(* IEC 61131-3 sources: fse/dataset/original (part 7) *)

(* ---- lb_claude_assisted_dd04b7ea0182_0007.st ---- *)
(*
This code implements a randomly grown symbolic expression:

((!(!(IN21 & (xor(xor(false, !(!((xor(xor(false, IN2), IN25)) | (!(IN9))))), ((IN33 & (xor(xor(IN17, IN40), IN11))) & (xor(xor(xor(xor(IN20, IN38), IN8), IN28 & IN33), IN19 & IN13))) & IN13))))) & IN25) & ((!((xor(xor(IN28, xor(xor((!(!(IN8 | IN21))) | ((!(IN47 | IN48)) | (!(IN15))), (!(IN9)) | ((xor(xor(IN49 & IN47, IN49 & IN24), IN46 | IN22)) | (!(IN28)))), !(((IN34 & IN44) & IN48) & IN26))), !(xor(xor(!((xor(xor(IN22, IN48), IN19)) | IN13), IN46), !((xor(xor(IN22, IN42), IN14)) | IN16))))) & ((((xor(xor((false | IN22) & (IN6 & IN36), (!(IN36)) & (IN1 & IN42)), IN21 & IN2)) | IN42) | IN48) | (!(IN36))))) & (IN15 | ((xor(xor(!(!(xor(xor((IN30 | IN11) | (IN43 & IN31), IN43 & (IN50 | IN12)), (IN13 & IN46) | (IN47 & IN18)))), ((IN47 | ((!(IN45)) & IN30)) & (xor(xor(xor(xor(IN6, IN1 & IN6), IN47), xor(xor(IN1 | IN29, IN33), false)), IN35))) | (xor(xor(((!(IN21)) | (!(IN25))) & (IN46 & (IN9 | IN19)), xor(xor(!(IN12 | IN11), xor(xor(IN8 & IN17, IN35 & IN20), xor(xor(IN38, IN14), IN18))), IN36 | (IN49 | IN43))), xor(xor((IN5 & IN20) & (xor(xor(IN20, IN17), IN15)), (xor(xor(IN2, IN24), IN37)) & IN6), IN18 & (IN41 | IN4))))), !(xor(xor(IN3, IN35), (xor(xor(IN29 & IN48, xor(xor(IN41, IN30), IN24)), IN15 | IN43)) | ((!(IN29)) | (false | IN42)))))) & (!(!(IN21 | (((!(IN38)) | (IN48 | IN49)) | IN16)))))))

*)

FUNCTION_BLOCK F_CollectInput
  VAR_IN_OUT
      Data : ARRAY[1..50] OF BOOL;
  END_VAR
  VAR_INPUT
      TICK  : BOOL := 0;
      IN1   : BOOL := 0;
      IN2   : BOOL := 0;
      IN3   : BOOL := 0;
      IN4   : BOOL := 0;
      IN5   : BOOL := 0;
      RESET : BOOL := FALSE;
  END_VAR
  VAR_OUTPUT
      Finished : BOOL;
  END_VAR
  VAR
      j    : USINT := 1;
      tock : BOOL  := 0;
  END_VAR
  IF NOT RESET AND tock = NOT TICK THEN
      Data[j]   := IN1;
      Data[j+1] := IN2;
      Data[j+2] := IN3;
      Data[j+3] := IN4;
      Data[j+4] := IN5;
      j := j + 5;
      tock := TICK;
  ELSE
      j := 1;
      tock := 0;
  END_IF;
  Finished := (j > 50);
END_FUNCTION_BLOCK

PROGRAM Boiler
  VAR
    Data  : ARRAY[1..50] OF BOOL;
    Ready : BOOL;
    CollectInput : F_CollectInput;
  END_VAR
  VAR
    TICK     AT %IX1.0 : BOOL;
    IN1      AT %IX0.3 : BOOL;
    IN2      AT %IX0.4 : BOOL;
    IN3      AT %IX0.5 : BOOL;
    IN4      AT %IX0.6 : BOOL;
    IN5      AT %IX0.7 : BOOL;
    OutReady AT %QX0.0 : BOOL := FALSE;
    FeedNext AT %QX0.1 : BOOL := FALSE;
    Out      AT %QX0.2 : BOOL;
  END_VAR
  CollectInput(TICK:=TICK, IN1:=IN1, IN2:=IN2, IN3:=IN3, IN4:=IN4, IN5:=IN5);
  Ready := CollectInput.Finished;
  FeedNext := 1;
  IF Ready THEN
    Out := (((NOT (NOT (Data[21] AND ((FALSE XOR (NOT (NOT (((FALSE XOR Data[2]) XOR Data[25]) OR (NOT Data[9]))))) XOR (((Data[33] AND ((Data[17] XOR Data[40]) XOR Data[11])) AND ((((Data[20] XOR Data[38]) XOR Data[8]) XOR (Data[28] AND Data[33])) XOR (Data[19] AND Data[13]))) AND Data[13]))))) AND Data[25]) AND ((NOT (((Data[28] XOR ((((NOT (NOT (Data[8] OR Data[21]))) OR ((NOT (Data[47] OR Data[48])) OR (NOT Data[15]))) XOR ((NOT Data[9]) OR ((((Data[49] AND Data[47]) XOR (Data[49] AND Data[24])) XOR (Data[46] OR Data[22])) OR (NOT Data[28])))) XOR (NOT (((Data[34] AND Data[44]) AND Data[48]) AND Data[26])))) XOR (NOT (((NOT (((Data[22] XOR Data[48]) XOR Data[19]) OR Data[13])) XOR Data[46]) XOR (NOT (((Data[22] XOR Data[42]) XOR Data[14]) OR Data[16]))))) AND (((((((FALSE OR Data[22]) AND (Data[6] AND Data[36])) XOR ((NOT Data[36]) AND (Data[1] AND Data[42]))) XOR (Data[21] AND Data[2])) OR Data[42]) OR Data[48]) OR (NOT Data[36])))) AND (Data[15] OR ((((NOT (NOT ((((Data[30] OR Data[11]) OR (Data[43] AND Data[31])) XOR (Data[43] AND (Data[50] OR Data[12]))) XOR ((Data[13] AND Data[46]) OR (Data[47] AND Data[18]))))) XOR (((Data[47] OR ((NOT Data[45]) AND Data[30])) AND ((((Data[6] XOR (Data[1] AND Data[6])) XOR Data[47]) XOR (((Data[1] OR Data[29]) XOR Data[33]) XOR FALSE)) XOR Data[35])) OR (((((NOT Data[21]) OR (NOT Data[25])) AND (Data[46] AND (Data[9] OR Data[19]))) XOR (((NOT (Data[12] OR Data[11])) XOR (((Data[8] AND Data[17]) XOR (Data[35] AND Data[20])) XOR ((Data[38] XOR Data[14]) XOR Data[18]))) XOR (Data[36] OR (Data[49] OR Data[43])))) XOR ((((Data[5] AND Data[20]) AND ((Data[20] XOR Data[17]) XOR Data[15])) XOR (((Data[2] XOR Data[24]) XOR Data[37]) AND Data[6])) XOR (Data[18] AND (Data[41] OR Data[4])))))) XOR (NOT ((Data[3] XOR Data[35]) XOR ((((Data[29] AND Data[48]) XOR ((Data[41] XOR Data[30]) XOR Data[24])) XOR (Data[15] OR Data[43])) OR ((NOT Data[29]) OR (FALSE OR Data[42])))))) AND (NOT (NOT (Data[21] OR (((NOT Data[38]) OR (Data[48] OR Data[49])) OR Data[16]))))))));
    OutReady := 1;
    CollectInput(RESET:=TRUE);
  END_IF;
END_PROGRAM

CONFIGURATION Config0
  RESOURCE Res0 ON PLC
    TASK task0(INTERVAL := T#20ms,PRIORITY := 0);
    PROGRAM instance0 WITH task0 : Boiler;
  END_RESOURCE
END_CONFIGURATION

(* ---- lb_claude_assisted_ddda264e743a_0020.st ---- *)
FUNCTION_BLOCK T_PLC_MS_block
	VAR_OUTPUT
		T_PLC_MS :	UDINT;
	END_VAR

	VAR_EXTERNAL
		PLC_TICKS_PER_SEC :	INT;
		PLC_SYS_TICK_CNT :	DINT;
	END_VAR

	VAR
		debug :	BOOL;(*Debug-Mode ON / OFF*)
		N :	INT;(*Debug-Faktor*)
		Offset :	UDINT;(*Debug-Offset*)
		temp :	DWORD := DWORD#1;(*Debug-Offset*)
		mode :	BOOL;(*modus*)
		faktor :	UDINT;(*Systemtakt-Faktor*)
		init :	BOOL;
		v_plc_ticks_per_sec :	UDINT;
		base :	UDINT := UDINT#1000;
	END_VAR

	IF init = FALSE THEN
		v_plc_ticks_per_sec := INT_TO_UDINT(PLC_TICKS_PER_SEC);
		IF v_plc_ticks_per_sec = UDINT#1024 THEN
			faktor := UDINT#1;
			mode := FALSE;
		ELSIF v_plc_ticks_per_sec > UDINT#0 THEN
			IF v_plc_ticks_per_sec <= base THEN
				faktor := base / v_plc_ticks_per_sec;
				mode := FALSE;
			ELSE
				faktor := v_plc_ticks_per_sec / base;
				mode := TRUE;
			END_IF;
		ELSE
			faktor := UDINT#1;
		END_IF;
		init := TRUE;
	END_IF;

	IF mode THEN
		T_PLC_MS := DINT_TO_UDINT(PLC_SYS_TICK_CNT) / faktor;
	ELSE
		T_PLC_MS := DINT_TO_UDINT(PLC_SYS_TICK_CNT) * faktor;
	END_IF;

	IF debug THEN
		T_PLC_MS := (DWORD_TO_UDINT(SHL(UDINT_TO_DWORD(T_PLC_MS),N) OR SHL(temp,N)) - UDINT#1) + Offset;
	END_IF;
END_FUNCTION_BLOCK

FUNCTION TIME_TO_UDINT2:UDINT
	VAR_INPUT
		X :	TIME;
	END_VAR

	TIME_TO_UDINT2 := DINT_TO_UDINT(TIME_TO_DINT(X));
END_FUNCTION

FUNCTION_BLOCK TUNE2_Block

	VAR_INPUT
		SET :	BOOL;
		SU :	BOOL;
		SD :	BOOL;
		FU :	BOOL;
		FD :	BOOL;
		RST :	BOOL;
		SS :	REAL := 0.1;
		FS :	REAL := 5.0;
		LIMIT_L :	REAL;
		LIMIT_H :	REAL := 100.0;
		RST_VAL :	REAL;
		SET_VAL :	REAL := 100.0;
		TR :	TIME := T#500ms;
		S1 :	REAL := 2.0;
		S2 :	REAL := 10.0;
	END_VAR

	VAR_OUTPUT
		Y :	REAL;
	END_VAR

	VAR
		tx :	UDINT;
		start :	UDINT;
		state :	INT;
		in :	BOOL;
		step2 :	REAL;
		speed :	REAL;
		Y_start :	REAL;
		T_PLC_MS :	T_PLC_MS_block;
	END_VAR

	T_PLC_MS();
	tx:= T_PLC_MS.T_PLC_MS;

	IF rst THEN
		Y := RST_val;
		state := 0;
	ELSIF set THEN
		Y := SET_val;
		state := 0;
	ELSIF state > 0 THEN
		CASE state OF
			1 :
				in := su;
			2 :
				in := sd;
			3 :
				in := fu;
			4 :
				in := fd;
		END_CASE;
		IF NOT in AND tx - start <= TIME_TO_UDINT2(TR) THEN
			Y := Y_start + step2;
			state := 0;
		ELSIF in AND tx - start >= TIME_TO_UDINT2(TR) THEN
			Y := Y_start + UDINT_TO_REAL(tx - start - TIME_TO_UDINT2(TR)) * speed;
		ELSIF NOT in THEN
			state := 0;
		END_IF;
	ELSIF su THEN
		state := 1;
		start := tx;
		step2 := ss;
		speed := s1 * 1.0E-3;
		Y_start := Y;
	ELSIF sd THEN
		state := 2;
		start := tx;
		step2 := -ss;
		speed := -s1 * 1.0E-3;
		Y_start := Y;
	ELSIF fu THEN
		state := 3;
		start := tx;
		step2 := fs;
		speed := s2 * 1.0E-3;
		y_start := Y;
	ELSIF fd THEN
		state := 4;
		start := tx;
		step2 := -fs;
		speed := -s2 * 1.0E-3;
		y_start := Y;
	END_IF;
END_FUNCTION_BLOCK

PROGRAM program0
  	VAR
		SET :	BOOL;
		SU :	BOOL;
		SD :	BOOL;
		FU :	BOOL;
		FD :	BOOL;
		RST :	BOOL;
		SS :	REAL;
		FS :	REAL;
		LIMIT_L :	REAL;
		LIMIT_H :	REAL;
		RST_VAL :	REAL;
		SET_VAL :	REAL;
		TR :	TIME ;
		S1 :	REAL;
		S2 :	REAL;
		Y :	REAL;
		func_block : TUNE2_Block;
  	END_VAR
	func_block.SET := SET;
	func_block.SU := SU;
	func_block.SD := SD;
	func_block.FU := FU;
	func_block.FD := FD;
	func_block.RST := RST;
	func_block.SS:= SS;
	func_block.FS := FS;
	func_block.LIMIT_L := LIMIT_L;
	func_block.LIMIT_H := LIMIT_H;
	func_block.RST_VAL := RST_VAL;
	func_block.SET_VAL := SET_VAL;
	func_block.TR := TR;
	func_block.S1 := S1;
	func_block.S2 := S2;
	func_block();
	Y := func_block.Y;
END_PROGRAM

CONFIGURATION Config0
	VAR_GLOBAL
		PLC_TICKS_PER_SEC :	INT;
		PLC_SYS_TICK_CNT :	DINT;
	END_VAR

	RESOURCE Res0 ON PLC
		TASK task0(INTERVAL := T#20ms,PRIORITY := 0);
		PROGRAM instance0 WITH task0 : program0;
	END_RESOURCE
END_CONFIGURATION

(* ---- lb_claude_assisted_def584e78dd9_0028.st ---- *)
(*
This code implements a randomly grown symbolic expression:

((xor(xor(!(IN17), IN3), IN42 & (!(!((!(xor(xor(IN42 & IN8, IN18), IN49))) | (!(IN32))))))) & ((!(!((IN47 | (IN12 & (xor(xor(!(IN9), IN41 & IN17), IN45)))) & (xor(xor(IN6 & (IN23 | (IN31 | IN44)), xor(xor((!(IN32)) & (!(IN23)), IN42 & (IN50 | IN34)), xor(xor(!(IN34), !(IN32)), IN15))), xor(xor(IN33, xor(xor(IN45 & IN5, IN11 & IN16), IN3 | IN4)), !(!(IN15)))))))) & (((xor(xor(((xor(xor(IN50 | IN14, IN46 & IN40), xor(xor(IN3, IN41), IN9))) & (IN22 & IN28)) | (xor(xor(IN41 | (IN26 & IN10), xor(xor(IN42 & IN12, xor(xor(IN32, IN46), IN35)), IN1 & IN11)), xor(xor(xor(xor(IN43, IN19), IN38), IN27 | IN21), !(IN10)))), !(xor(xor((xor(xor(IN7, IN50), IN1)) | IN6, (IN35 & IN3) | (!(IN28))), xor(xor(IN7 & IN16, IN37 | IN33), IN11)))), (!((!(IN25)) | (!(IN41)))) & ((!(IN33 & true)) & (!(!(IN5)))))) & (xor(xor(IN12, !(IN17)), (((!(IN28)) & (xor(xor(IN4, IN22), IN12))) | ((IN4 & IN38) & IN37)) | true))) | IN6))) & (xor(xor(!(IN24), xor(xor(!((xor(xor(IN48 | (!((IN17 & IN14) | IN31)), (xor(xor(true, xor(xor(xor(xor(IN16, IN16), IN17), !(IN23)), IN2)), (!(IN45)) | (xor(xor(IN31, IN48), IN25)))) & (!(xor(xor(IN6, IN41 & IN37), IN38)))), (IN26 | ((IN7 & IN2) | (IN17 | false))) & (xor(xor(IN42 & (IN28 | IN44), (IN16 & IN26) | (IN21 | IN13)), (IN11 & IN4) | (IN48 | IN47))))) & ((!(false & ((xor(xor(IN20, IN8), IN2)) | (IN36 & IN18)))) & IN47)), xor(xor(((false & (xor(xor(xor(xor(IN27 | IN30, xor(xor(IN23, IN27), IN7)), IN21), !(IN50)), (!(IN35)) & (xor(xor(IN21, IN7), IN17))))) | ((((IN9 | IN5) | (xor(xor(IN46, IN31), IN33))) | IN14) | IN32)) | (((!(IN19)) & IN21) & (!((!(IN44 & IN26)) | IN42))), xor(xor(!(IN34), (IN31 | (xor(xor(IN20, IN9), IN30))) | (xor(xor(IN21, xor(xor((IN29 | IN5) | (IN10 & IN14), xor(xor(IN41 & IN34, xor(xor(IN20, IN4), IN29)), IN29 & IN17)), IN39 | (IN7 & IN43))), ((!(IN40)) | IN50) | (!(IN17))))), xor(xor(xor(xor(IN31, IN24), ((IN30 | IN5) & (!(IN48))) | ((xor(xor(IN16, IN13), IN34)) & (!(IN16)))), (xor(xor(IN29 | IN25, xor(xor(xor(xor(IN20, IN40), IN9), IN26 | IN20), IN43 | IN32)), (xor(xor(IN35, IN6), IN33)) | (IN30 | IN7))) & (((true | IN15) | (IN46 | IN5)) | ((xor(xor(IN20, IN39), IN5)) | (IN48 | IN20)))), ((!(IN11 & IN1)) | ((xor(xor(IN5, IN25), IN49)) | (IN3 & IN43))) | (!(xor(xor(IN22, xor(xor(IN40, IN26), IN7)), xor(xor(IN10, IN10), IN44))))))), !(xor(xor(!(xor(xor((!(IN32)) | (xor(xor(IN28, IN4), IN11)), (IN7 | IN49) & (IN19 | IN17)), xor(xor(xor(xor(IN50, IN4), IN7), !(IN25)), !(IN10)))), (xor(xor(IN18 & (IN23 | IN36), xor(xor(IN36 | false, IN31 | IN19), IN15 & IN5)), !(IN41))) | (!(!(xor(xor(IN34, IN8), true))))), IN10 & (((IN39 & IN8) | (xor(xor(IN37, IN1), IN46))) | ((xor(xor(IN21, IN1), IN16)) | (false | IN1))))))), IN25 & (IN31 & (IN20 & IN46)))), IN38 | (!(IN32))))

*)

FUNCTION_BLOCK F_CollectInput
  VAR_IN_OUT
      Data : ARRAY[1..50] OF BOOL;
  END_VAR
  VAR_INPUT
      TICK  : BOOL := 0;
      IN1   : BOOL := 0;
      IN2   : BOOL := 0;
      IN3   : BOOL := 0;
      IN4   : BOOL := 0;
      IN5   : BOOL := 0;
      RESET : BOOL := FALSE;
  END_VAR
  VAR_OUTPUT
      Finished : BOOL;
  END_VAR
  VAR
      j    : USINT := 1;
      tock : BOOL  := 0;
  END_VAR
  IF NOT RESET AND tock = NOT TICK THEN
      Data[j]   := IN1;
      Data[j+1] := IN2;
      Data[j+2] := IN3;
      Data[j+3] := IN4;
      Data[j+4] := IN5;
      j := j + 5;
      tock := TICK;
  ELSE
      j := 1;
      tock := 0;
  END_IF;
  Finished := (j > 50);
END_FUNCTION_BLOCK

PROGRAM Boiler
  VAR
    Data  : ARRAY[1..50] OF BOOL;
    Ready : BOOL;
    CollectInput : F_CollectInput;
  END_VAR
  VAR
    TICK     AT %IX1.0 : BOOL;
    IN1      AT %IX0.3 : BOOL;
    IN2      AT %IX0.4 : BOOL;
    IN3      AT %IX0.5 : BOOL;
    IN4      AT %IX0.6 : BOOL;
    IN5      AT %IX0.7 : BOOL;
    OutReady AT %QX0.0 : BOOL := FALSE;
    FeedNext AT %QX0.1 : BOOL := FALSE;
    Out      AT %QX0.2 : BOOL;
  END_VAR
  CollectInput(TICK:=TICK, IN1:=IN1, IN2:=IN2, IN3:=IN3, IN4:=IN4, IN5:=IN5);
  Ready := CollectInput.Finished;
  FeedNext := 1;
  IF Ready THEN
    Out := (((((NOT Data[17]) XOR Data[3]) XOR (Data[42] AND (NOT (NOT ((NOT (((Data[42] AND Data[8]) XOR Data[18]) XOR Data[49])) OR (NOT Data[32])))))) AND ((NOT (NOT ((Data[47] OR (Data[12] AND (((NOT Data[9]) XOR (Data[41] AND Data[17])) XOR Data[45]))) AND (((Data[6] AND (Data[23] OR (Data[31] OR Data[44]))) XOR ((((NOT Data[32]) AND (NOT Data[23])) XOR (Data[42] AND (Data[50] OR Data[34]))) XOR (((NOT Data[34]) XOR (NOT Data[32])) XOR Data[15]))) XOR ((Data[33] XOR (((Data[45] AND Data[5]) XOR (Data[11] AND Data[16])) XOR (Data[3] OR Data[4]))) XOR (NOT (NOT Data[15]))))))) AND (((((((((Data[50] OR Data[14]) XOR (Data[46] AND Data[40])) XOR ((Data[3] XOR Data[41]) XOR Data[9])) AND (Data[22] AND Data[28])) OR (((Data[41] OR (Data[26] AND Data[10])) XOR (((Data[42] AND Data[12]) XOR ((Data[32] XOR Data[46]) XOR Data[35])) XOR (Data[1] AND Data[11]))) XOR ((((Data[43] XOR Data[19]) XOR Data[38]) XOR (Data[27] OR Data[21])) XOR (NOT Data[10])))) XOR (NOT (((((Data[7] XOR Data[50]) XOR Data[1]) OR Data[6]) XOR ((Data[35] AND Data[3]) OR (NOT Data[28]))) XOR (((Data[7] AND Data[16]) XOR (Data[37] OR Data[33])) XOR Data[11])))) XOR ((NOT ((NOT Data[25]) OR (NOT Data[41]))) AND ((NOT (Data[33] AND TRUE)) AND (NOT (NOT Data[5]))))) AND ((Data[12] XOR (NOT Data[17])) XOR ((((NOT Data[28]) AND ((Data[4] XOR Data[22]) XOR Data[12])) OR ((Data[4] AND Data[38]) AND Data[37])) OR TRUE))) OR Data[6]))) AND (((NOT Data[24]) XOR (((NOT ((((Data[48] OR (NOT ((Data[17] AND Data[14]) OR Data[31]))) XOR (((TRUE XOR ((((Data[16] XOR Data[16]) XOR Data[17]) XOR (NOT Data[23])) XOR Data[2])) XOR ((NOT Data[45]) OR ((Data[31] XOR Data[48]) XOR Data[25]))) AND (NOT ((Data[6] XOR (Data[41] AND Data[37])) XOR Data[38])))) XOR ((Data[26] OR ((Data[7] AND Data[2]) OR (Data[17] OR FALSE))) AND (((Data[42] AND (Data[28] OR Data[44])) XOR ((Data[16] AND Data[26]) OR (Data[21] OR Data[13]))) XOR ((Data[11] AND Data[4]) OR (Data[48] OR Data[47]))))) AND ((NOT (FALSE AND (((Data[20] XOR Data[8]) XOR Data[2]) OR (Data[36] AND Data[18])))) AND Data[47]))) XOR (((((FALSE AND (((((Data[27] OR Data[30]) XOR ((Data[23] XOR Data[27]) XOR Data[7])) XOR Data[21]) XOR (NOT Data[50])) XOR ((NOT Data[35]) AND ((Data[21] XOR Data[7]) XOR Data[17])))) OR ((((Data[9] OR Data[5]) OR ((Data[46] XOR Data[31]) XOR Data[33])) OR Data[14]) OR Data[32])) OR (((NOT Data[19]) AND Data[21]) AND (NOT ((NOT (Data[44] AND Data[26])) OR Data[42])))) XOR (((NOT Data[34]) XOR ((Data[31] OR ((Data[20] XOR Data[9]) XOR Data[30])) OR ((Data[21] XOR ((((Data[29] OR Data[5]) OR (Data[10] AND Data[14])) XOR (((Data[41] AND Data[34]) XOR ((Data[20] XOR Data[4]) XOR Data[29])) XOR (Data[29] AND Data[17]))) XOR (Data[39] OR (Data[7] AND Data[43])))) XOR (((NOT Data[40]) OR Data[50]) OR (NOT Data[17]))))) XOR ((((Data[31] XOR Data[24]) XOR (((Data[30] OR Data[5]) AND (NOT Data[48])) OR (((Data[16] XOR Data[13]) XOR Data[34]) AND (NOT Data[16])))) XOR ((((Data[29] OR Data[25]) XOR ((((Data[20] XOR Data[40]) XOR Data[9]) XOR (Data[26] OR Data[20])) XOR (Data[43] OR Data[32]))) XOR (((Data[35] XOR Data[6]) XOR Data[33]) OR (Data[30] OR Data[7]))) AND (((TRUE OR Data[15]) OR (Data[46] OR Data[5])) OR (((Data[20] XOR Data[39]) XOR Data[5]) OR (Data[48] OR Data[20]))))) XOR (((NOT (Data[11] AND Data[1])) OR (((Data[5] XOR Data[25]) XOR Data[49]) OR (Data[3] AND Data[43]))) OR (NOT ((Data[22] XOR ((Data[40] XOR Data[26]) XOR Data[7])) XOR ((Data[10] XOR Data[10]) XOR Data[44]))))))) XOR (NOT (((NOT ((((NOT Data[32]) OR ((Data[28] XOR Data[4]) XOR Data[11])) XOR ((Data[7] OR Data[49]) AND (Data[19] OR Data[17]))) XOR ((((Data[50] XOR Data[4]) XOR Data[7]) XOR (NOT Data[25])) XOR (NOT Data[10])))) XOR ((((Data[18] AND (Data[23] OR Data[36])) XOR (((Data[36] OR FALSE) XOR (Data[31] OR Data[19])) XOR (Data[15] AND Data[5]))) XOR (NOT Data[41])) OR (NOT (NOT ((Data[34] XOR Data[8]) XOR TRUE))))) XOR (Data[10] AND (((Data[39] AND Data[8]) OR ((Data[37] XOR Data[1]) XOR Data[46])) OR (((Data[21] XOR Data[1]) XOR Data[16]) OR (FALSE OR Data[1])))))))) XOR (Data[25] AND (Data[31] AND (Data[20] AND Data[46]))))) XOR (Data[38] OR (NOT Data[32]))));
    OutReady := 1;
    CollectInput(RESET:=TRUE);
  END_IF;
END_PROGRAM

CONFIGURATION Config0
  RESOURCE Res0 ON PLC
    TASK task0(INTERVAL := T#20ms,PRIORITY := 0);
    PROGRAM instance0 WITH task0 : Boiler;
  END_RESOURCE
END_CONFIGURATION

(* ---- lb_claude_assisted_df27abd0aee2_0074.st ---- *)
FUNCTION_BLOCK EQ_0
  VAR_INPUT
    IN1 : DINT;
    IN2 : DINT;
  END_VAR
  VAR_OUTPUT
    OUT : BOOL;
  END_VAR
  VAR
    i : INT;
    mytimer : TON;
  END_VAR

  OUT:=FALSE;
  IF IN1=IN2 then
    OUT:=TRUE;
  END_IF;

  mytimer(IN := TRUE, PT := t#8000ms);
  i:=0;
  IF mytimer.Q = TRUE then
     WHILE i<4 do
      OUT:=TRUE;
    End_WHILE;
  End_IF;

END_FUNCTION_BLOCK

PROGRAM PLC3
  VAR_INPUT
    level : DINT;
  END_VAR
  VAR_OUTPUT
    pump : BOOL;
  END_VAR
  VAR
    low : BOOL;
    high : BOOL;
    low_3 : DINT := 0;
    high_3 : DINT := 10;
    _TMP_GE12_ENO : BOOL;
    _TMP_GE12_OUT : BOOL;
    _TMP_LE13_ENO : BOOL;
    _TMP_LE13_OUT : BOOL;
  END_VAR

  _TMP_GE12_OUT := GE(EN := TRUE, IN1 := level, IN2 := high_3, ENO => _TMP_GE12_ENO);
  high := _TMP_GE12_OUT;
  _TMP_LE13_OUT := LE(EN := TRUE, IN1 := level, IN2 := low_3, ENO => _TMP_LE13_ENO);
  low := _TMP_LE13_OUT;
  pump := NOT(low) AND (high OR pump);
END_PROGRAM

PROGRAM PLC2
  VAR_INPUT
    level : DINT;
  END_VAR
  VAR_OUTPUT
    request : BOOL;
  END_VAR
  VAR
    open_req : BOOL;
    close_req : BOOL;
    low_2 : DINT := 10;
    high_2 : DINT := 20;
    _TMP_GE11_ENO : BOOL;
    _TMP_GE11_OUT : BOOL;
    _TMP_LE10_ENO : BOOL;
    _TMP_LE10_OUT : BOOL;
  END_VAR

  _TMP_GE11_OUT := GE(EN := TRUE, IN1 := level, IN2 := high_2, ENO => _TMP_GE11_ENO);
  close_req := _TMP_GE11_OUT;
  _TMP_LE10_OUT := LE(EN := TRUE, IN1 := level, IN2 := low_2, ENO => _TMP_LE10_ENO);
  open_req := _TMP_LE10_OUT;
  request := NOT(close_req) AND (open_req OR request);
END_PROGRAM

PROGRAM PLC1
  VAR_INPUT
    level : DINT;
    request : DINT;
  END_VAR
  VAR_OUTPUT
    pumps : BOOL;
    valve : BOOL;
  END_VAR
  VAR
    low : BOOL;
    high : BOOL;
    open_req : BOOL;
    close_req : BOOL;
    low_1 : DINT := 40;
    high_1 : DINT := 80;
    EQ_00 : EQ_0;
    _TMP_EQ24_ENO : BOOL;
    _TMP_EQ24_OUT : BOOL;
    _TMP_LE3_ENO : BOOL;
    _TMP_LE3_OUT : BOOL;
    _TMP_GE7_ENO : BOOL;
    _TMP_GE7_OUT : BOOL;
  END_VAR

  EQ_00(EN := TRUE, IN1 := request, IN2 := 1);
  open_req := EQ_00.OUT;
  _TMP_EQ24_OUT := EQ(EN := TRUE, IN1 := request, IN2 := 0, ENO => _TMP_EQ24_ENO);
  close_req := _TMP_EQ24_OUT;
  pumps := NOT(high) AND (low OR pumps);
  valve := NOT(close_req) AND (valve OR open_req AND NOT(low));
  _TMP_LE3_OUT := LE(EN := TRUE, IN1 := level, IN2 := low_1, ENO => _TMP_LE3_ENO);
  low := _TMP_LE3_OUT;
  _TMP_GE7_OUT := GE(EN := TRUE, IN1 := level, IN2 := high_1, ENO => _TMP_GE7_ENO);
  high := _TMP_GE7_OUT;
END_PROGRAM

CONFIGURATION Config0

  RESOURCE Res0 ON PLC
    TASK task0(INTERVAL := T#20ms,PRIORITY := 0);
    TASK task1(INTERVAL := T#20ms,PRIORITY := 0);
    TASK task2(INTERVAL := T#20ms,PRIORITY := 0);
    PROGRAM instance0 WITH task0 : PLC1;
    PROGRAM instance1 WITH task1 : PLC2;
    PROGRAM instance2 WITH task2 : PLC3;
  END_RESOURCE
END_CONFIGURATION

(* ---- lb_claude_assisted_e1afd5a5507c_0051.st ---- *)
(*
This code implements a randomly grown symbolic expression:

(IN29 | (((!(IN27)) | (xor(xor(!(xor(xor(!((!(IN8)) & IN9), xor(xor(xor(xor(xor(xor(IN14, IN9), IN41), xor(xor(IN8, IN28), false)), xor(xor(IN9, IN9), IN2)), !(xor(xor(IN2, IN5), IN41))), (!(IN28)) & (xor(xor(IN12, IN39), IN7)))), IN36)), xor(xor(true, !(((IN30 | IN20) | IN9) & IN3)), xor(xor(false, (!(IN31)) | (xor(xor(IN41 | IN5, IN49 & IN1), !(IN13)))), xor(xor((IN28 | IN50) | (!(IN16)), (xor(xor(IN42, IN4), IN6)) | (xor(xor(IN38, IN42), IN36))), (xor(xor(IN46, IN18), IN35)) & (IN39 & IN11))))), IN39))) & (!(xor(xor(IN22 | ((!(xor(xor(IN21, IN5), IN41 & IN1))) | (xor(xor(xor(xor(IN15 | IN13, IN38 | IN6), !(IN1)), IN29), IN48))), IN18), IN3))))) | (!(!((((IN22 | (xor(xor(!(xor(xor(IN30, false), IN5)), !(IN14 | IN3)), !(IN48)))) | ((((!(IN28)) & (xor(xor(IN29, IN6), IN15))) & ((IN8 & IN49) | IN23)) & (((IN12 & IN1) | (xor(xor(IN43, IN5), IN47))) & ((!(IN33)) | (true | IN20))))) & ((!(IN50 | (!(IN5 | IN30)))) & IN40)) & (xor(xor((xor(xor((xor(xor(xor(xor(IN22, IN30), IN10), IN50), IN23 | IN47)) | (IN1 & (xor(xor(IN46, IN29), IN24))), IN24), ((IN2 & IN18) | (IN26 | IN47)) | ((!(IN19)) & IN35))) | ((IN33 & (!(IN25 | IN20))) | (xor(xor((xor(xor(IN40, IN13), IN19)) & (xor(xor(IN2, IN37), IN10)), (IN49 | IN40) & IN19), (xor(xor(IN25, IN24), IN14)) & (IN22 & IN32)))), (!(!((xor(xor(IN42, IN8), IN1)) & (!(IN42))))) & ((!(IN23 & IN19)) | ((!(IN29 & IN50)) & (!(IN8 & IN35))))), !(xor(xor(xor(xor((IN29 & IN22) & (!(IN14)), (IN32 & IN20) & (xor(xor(IN7, IN24), IN7))), (true & IN45) | (IN31 | IN44)), (xor(xor(!(IN45), IN35 | IN9), IN40 | IN3)) | ((xor(xor(IN5, IN37), IN27)) | (xor(xor(IN25, IN45), IN32)))), (false & (IN9 | IN18)) | (xor(xor(IN8, xor(xor(IN10, IN26), IN25)), !(IN39))))))))))

*)

FUNCTION_BLOCK F_CollectInput
  VAR_IN_OUT
      Data : ARRAY[1..50] OF BOOL;
  END_VAR
  VAR_INPUT
      TICK  : BOOL := 0;
      IN1   : BOOL := 0;
      IN2   : BOOL := 0;
      IN3   : BOOL := 0;
      IN4   : BOOL := 0;
      IN5   : BOOL := 0;
      RESET : BOOL := FALSE;
  END_VAR
  VAR_OUTPUT
      Finished : BOOL;
  END_VAR
  VAR
      j    : USINT := 1;
      tock : BOOL  := 0;
  END_VAR
  IF NOT RESET AND tock = NOT TICK THEN
      Data[j]   := IN1;
      Data[j+1] := IN2;
      Data[j+2] := IN3;
      Data[j+3] := IN4;
      Data[j+4] := IN5;
      j := j + 5;
      tock := TICK;
  ELSE
      j := 1;
      tock := 0;
  END_IF;
  Finished := (j > 50);
END_FUNCTION_BLOCK

PROGRAM Boiler
  VAR
    Data  : ARRAY[1..50] OF BOOL;
    Ready : BOOL;
    CollectInput : F_CollectInput;
  END_VAR
  VAR
    TICK     AT %IX1.0 : BOOL;
    IN1      AT %IX0.3 : BOOL;
    IN2      AT %IX0.4 : BOOL;
    IN3      AT %IX0.5 : BOOL;
    IN4      AT %IX0.6 : BOOL;
    IN5      AT %IX0.7 : BOOL;
    OutReady AT %QX0.0 : BOOL := FALSE;
    FeedNext AT %QX0.1 : BOOL := FALSE;
    Out      AT %QX0.2 : BOOL;
  END_VAR
  CollectInput(TICK:=TICK, IN1:=IN1, IN2:=IN2, IN3:=IN3, IN4:=IN4, IN5:=IN5);
  Ready := CollectInput.Finished;
  FeedNext := 1;
  IF Ready THEN
    Out := ((Data[29] OR (((NOT Data[27]) OR (((NOT (((NOT ((NOT Data[8]) AND Data[9])) XOR ((((((Data[14] XOR Data[9]) XOR Data[41]) XOR ((Data[8] XOR Data[28]) XOR FALSE)) XOR ((Data[9] XOR Data[9]) XOR Data[2])) XOR (NOT ((Data[2] XOR Data[5]) XOR Data[41]))) XOR ((NOT Data[28]) AND ((Data[12] XOR Data[39]) XOR Data[7])))) XOR Data[36])) XOR ((TRUE XOR (NOT (((Data[30] OR Data[20]) OR Data[9]) AND Data[3]))) XOR ((FALSE XOR ((NOT Data[31]) OR (((Data[41] OR Data[5]) XOR (Data[49] AND Data[1])) XOR (NOT Data[13])))) XOR ((((Data[28] OR Data[50]) OR (NOT Data[16])) XOR (((Data[42] XOR Data[4]) XOR Data[6]) OR ((Data[38] XOR Data[42]) XOR Data[36]))) XOR (((Data[46] XOR Data[18]) XOR Data[35]) AND (Data[39] AND Data[11])))))) XOR Data[39])) AND (NOT (((Data[22] OR ((NOT ((Data[21] XOR Data[5]) XOR (Data[41] AND Data[1]))) OR (((((Data[15] OR Data[13]) XOR (Data[38] OR Data[6])) XOR (NOT Data[1])) XOR Data[29]) XOR Data[48]))) XOR Data[18]) XOR Data[3])))) OR (NOT (NOT ((((Data[22] OR (((NOT ((Data[30] XOR FALSE) XOR Data[5])) XOR (NOT (Data[14] OR Data[3]))) XOR (NOT Data[48]))) OR ((((NOT Data[28]) AND ((Data[29] XOR Data[6]) XOR Data[15])) AND ((Data[8] AND Data[49]) OR Data[23])) AND (((Data[12] AND Data[1]) OR ((Data[43] XOR Data[5]) XOR Data[47])) AND ((NOT Data[33]) OR (TRUE OR Data[20]))))) AND ((NOT (Data[50] OR (NOT (Data[5] OR Data[30])))) AND Data[40])) AND ((((((((((Data[22] XOR Data[30]) XOR Data[10]) XOR Data[50]) XOR (Data[23] OR Data[47])) OR (Data[1] AND ((Data[46] XOR Data[29]) XOR Data[24]))) XOR Data[24]) XOR (((Data[2] AND Data[18]) OR (Data[26] OR Data[47])) OR ((NOT Data[19]) AND Data[35]))) OR ((Data[33] AND (NOT (Data[25] OR Data[20]))) OR (((((Data[40] XOR Data[13]) XOR Data[19]) AND ((Data[2] XOR Data[37]) XOR Data[10])) XOR ((Data[49] OR Data[40]) AND Data[19])) XOR (((Data[25] XOR Data[24]) XOR Data[14]) AND (Data[22] AND Data[32]))))) XOR ((NOT (NOT (((Data[42] XOR Data[8]) XOR Data[1]) AND (NOT Data[42])))) AND ((NOT (Data[23] AND Data[19])) OR ((NOT (Data[29] AND Data[50])) AND (NOT (Data[8] AND Data[35])))))) XOR (NOT ((((((Data[29] AND Data[22]) AND (NOT Data[14])) XOR ((Data[32] AND Data[20]) AND ((Data[7] XOR Data[24]) XOR Data[7]))) XOR ((TRUE AND Data[45]) OR (Data[31] OR Data[44]))) XOR ((((NOT Data[45]) XOR (Data[35] OR Data[9])) XOR (Data[40] OR Data[3])) OR (((Data[5] XOR Data[37]) XOR Data[27]) OR ((Data[25] XOR Data[45]) XOR Data[32])))) XOR ((FALSE AND (Data[9] OR Data[18])) OR ((Data[8] XOR ((Data[10] XOR Data[26]) XOR Data[25])) XOR (NOT Data[39]))))))))));
    OutReady := 1;
    CollectInput(RESET:=TRUE);
  END_IF;
END_PROGRAM

CONFIGURATION Config0
  RESOURCE Res0 ON PLC
    TASK task0(INTERVAL := T#20ms,PRIORITY := 0);
    PROGRAM instance0 WITH task0 : Boiler;
  END_RESOURCE
END_CONFIGURATION

(* ---- lb_claude_assisted_e232be441ee1_0058.st ---- *)
(*
This code implements a randomly grown symbolic expression:

(!(false & IN38)) & (!(IN32))

*)

FUNCTION_BLOCK F_CollectInput
  VAR_IN_OUT
      Data : ARRAY[1..50] OF BOOL;
  END_VAR
  VAR_INPUT
      TICK  : BOOL := 0;
      IN1   : BOOL := 0;
      IN2   : BOOL := 0;
      IN3   : BOOL := 0;
      IN4   : BOOL := 0;
      IN5   : BOOL := 0;
      RESET : BOOL := FALSE;
  END_VAR
  VAR_OUTPUT
      Finished : BOOL;
  END_VAR
  VAR
      j    : USINT := 1;
      tock : BOOL  := 0;
  END_VAR
  IF NOT RESET AND tock = NOT TICK THEN
      Data[j]   := IN1;
      Data[j+1] := IN2;
      Data[j+2] := IN3;
      Data[j+3] := IN4;
      Data[j+4] := IN5;
      j := j + 5;
      tock := TICK;
  ELSE
      j := 1;
      tock := 0;
  END_IF;
  Finished := (j > 50);
END_FUNCTION_BLOCK

PROGRAM Boiler
  VAR
    Data  : ARRAY[1..50] OF BOOL;
    Ready : BOOL;
    CollectInput : F_CollectInput;
  END_VAR
  VAR
    TICK     AT %IX1.0 : BOOL;
    IN1      AT %IX0.3 : BOOL;
    IN2      AT %IX0.4 : BOOL;
    IN3      AT %IX0.5 : BOOL;
    IN4      AT %IX0.6 : BOOL;
    IN5      AT %IX0.7 : BOOL;
    OutReady AT %QX0.0 : BOOL := FALSE;
    FeedNext AT %QX0.1 : BOOL := FALSE;
    Out      AT %QX0.2 : BOOL;
  END_VAR
  CollectInput(TICK:=TICK, IN1:=IN1, IN2:=IN2, IN3:=IN3, IN4:=IN4, IN5:=IN5);
  Ready := CollectInput.Finished;
  FeedNext := 1;
  IF Ready THEN
    Out := ((NOT (FALSE AND Data[38])) AND (NOT Data[32]));
    OutReady := 1;
    CollectInput(RESET:=TRUE);
  END_IF;
END_PROGRAM

CONFIGURATION Config0
  RESOURCE Res0 ON PLC
    TASK task0(INTERVAL := T#20ms,PRIORITY := 0);
    PROGRAM instance0 WITH task0 : Boiler;
  END_RESOURCE
END_CONFIGURATION

(* ---- lb_claude_assisted_e35f32df2f8c_0082.st ---- *)
FUNCTION_BLOCK T_PLC_MS_block
	VAR_OUTPUT
		T_PLC_MS :	UDINT;
	END_VAR

	VAR
		PLC_TICKS_PER_SEC :	INT;
		PLC_SYS_TICK_CNT :	DINT;
	END_VAR

	VAR
		debug :	BOOL;(*Debug-Mode ON / OFF*)
		N :	INT;(*Debug-Faktor*)
		Offset :	UDINT;(*Debug-Offset*)
		temp :	DWORD := DWORD#1;(*Debug-Offset*)
		MODE :	BOOL;(*modus*)
		faktor :	UDINT;(*Systemtakt-Faktor*)
		init :	BOOL;
		v_plc_ticks_per_sec :	UDINT;
		base :	UDINT := UDINT#1000;
	END_VAR

	IF init = FALSE THEN
		v_plc_ticks_per_sec := INT_TO_UDINT(PLC_TICKS_PER_SEC);
		IF v_plc_ticks_per_sec = UDINT#1024 THEN
			faktor := UDINT#1;
			MODE := FALSE;
		ELSIF v_plc_ticks_per_sec > UDINT#0 THEN
			IF v_plc_ticks_per_sec <= base THEN
				faktor := base / v_plc_ticks_per_sec;
				MODE := FALSE;
			ELSE
				faktor := v_plc_ticks_per_sec / base;
				MODE := TRUE;
			END_IF;
		ELSE
			faktor := UDINT#1;
		END_IF;
		init := TRUE;
	END_IF;

	IF MODE THEN
		T_PLC_MS := DINT_TO_UDINT(PLC_SYS_TICK_CNT) / faktor;
	ELSE
		T_PLC_MS := DINT_TO_UDINT(PLC_SYS_TICK_CNT) * faktor;
	END_IF;

	IF debug THEN
		T_PLC_MS := (DWORD_TO_UDINT(SHL(UDINT_TO_DWORD(T_PLC_MS),N) OR SHL(temp,N)) - UDINT#1) + Offset;
	END_IF;
END_FUNCTION_BLOCK

FUNCTION_BLOCK INTEGRATE

	VAR_INPUT
		E :	BOOL := TRUE;
		X :	REAL;
		K :	REAL := 1.0;
	END_VAR

	VAR_IN_OUT
		Y :	REAL;
	END_VAR

	VAR
		X_LAST :	REAL;
		init :	BOOL;
		T_PLC_MS :	T_PLC_MS_block;
		last :	UDINT;
		TX :	UDINT;
	END_VAR

	T_PLC_MS();
	TX:= T_PLC_MS.T_PLC_MS;

	IF NOT init THEN
		init := TRUE;
		X_LAST := X;
	ELSIF E THEN
		Y := (X + X_LAST) * 0.5E-3 * UDINT_TO_REAL(TX-last) * K + Y;
		X_LAST := X;
	END_IF;
	last := TX;

END_FUNCTION_BLOCK

FUNCTION_BLOCK FT_PT2

	VAR_INPUT
		IN :	REAL;
		T :	TIME;
		D :	REAL;
		K :	REAL := 1.0;
	END_VAR

	VAR_OUTPUT
		OUT :	REAL;
	END_VAR

	VAR
		init :	BOOL;
		int1 :	INTEGRATE;
		int2 :	INTEGRATE;
		TN :	REAL;
		I1 :	REAL;
		I2 :	REAL;
		tn2 :	REAL;
	END_VAR

	IF NOT init OR T = T#0s THEN
		init := TRUE;
		OUT := K * IN;
		I2 := OUT;
	ELSE
		TN := TIME_TO_REAL(T) / 1000.0;
		tn2 := TN * TN;
		int1(X := IN * K / tn2 - I1 * 0.5 * D / TN - I2 / tn2, Y := I1);
		I1 := int1.Y;
		int2(X := I1,Y := I2);
		I2 := int2.Y;
		OUT := I2;
	END_IF;

END_FUNCTION_BLOCK

PROGRAM program0
	VAR
		IN :	REAL;
		T :	TIME;
		D :	REAL;
		K :	REAL := 1.0;

		OUT :	REAL;

		func_block : FT_PT2;
	END_VAR
	func_block.IN := IN;
	func_block.T := T;
	func_block.D := D;
	func_block.K := K;
	func_block();
	OUT := func_block.OUT;
END_PROGRAM

(* ---- lb_claude_assisted_e419d39d0817_0009.st ---- *)
TYPE
  LOGLEVEL : (CRITICAL, WARNING, INFO, DEBUG) := INFO;
END_TYPE

FUNCTION_BLOCK LOGGER
  VAR_INPUT
    TRIG : BOOL;
    MSG : STRING;
    LEVEL : LOGLEVEL := INFO;
  END_VAR
  VAR
    TRIG0 : BOOL;
  END_VAR

  IF TRIG AND NOT TRIG0 THEN
  {{
   LogMessage(GetFbVar(LEVEL),(char*)GetFbVar(MSG, .body),GetFbVar(MSG, .len));
  }}
  END_IF;
  TRIG0:=TRIG;
END_FUNCTION_BLOCK

FUNCTION_BLOCK python_eval
  VAR_INPUT
    TRIG : BOOL;
    CODE : STRING;
  END_VAR
  VAR_OUTPUT
    ACK : BOOL;
    RESULT : STRING;
  END_VAR
  VAR
    STATE : DWORD;
    BUFFER : STRING;
    PREBUFFER : STRING;
    TRIGM1 : BOOL;
    TRIGGED : BOOL;
  END_VAR

  {extern void __PythonEvalFB(int, PYTHON_EVAL*);__PythonEvalFB(0, data__);}
END_FUNCTION_BLOCK

FUNCTION_BLOCK python_poll
  VAR_INPUT
    TRIG : BOOL;
    CODE : STRING;
  END_VAR
  VAR_OUTPUT
    ACK : BOOL;
    RESULT : STRING;
  END_VAR
  VAR
    STATE : DWORD;
    BUFFER : STRING;
    PREBUFFER : STRING;
    TRIGM1 : BOOL;
    TRIGGED : BOOL;
  END_VAR

  {extern void __PythonEvalFB(int, PYTHON_EVAL*);__PythonEvalFB(1,(PYTHON_EVAL*)(void*)data__);}
END_FUNCTION_BLOCK

FUNCTION_BLOCK python_gear
  VAR_INPUT
    N : UINT;
    TRIG : BOOL;
    CODE : STRING;
  END_VAR
  VAR_OUTPUT
    ACK : BOOL;
    RESULT : STRING;
  END_VAR
  VAR
    py_eval : python_eval;
    COUNTER : UINT;
    ADD10_OUT : UINT;
    EQ13_OUT : BOOL;
    SEL15_OUT : UINT;
    AND7_OUT : BOOL;
  END_VAR

  ADD10_OUT := ADD(COUNTER, 1);
  EQ13_OUT := EQ(N, ADD10_OUT);
  SEL15_OUT := SEL(EQ13_OUT, ADD10_OUT, 0);
  COUNTER := SEL15_OUT;
  AND7_OUT := AND(EQ13_OUT, TRIG);
  py_eval(TRIG := AND7_OUT, CODE := CODE);
  ACK := py_eval.ACK;
  RESULT := py_eval.RESULT;
END_FUNCTION_BLOCK

FUNCTION TEMP_NI : REAL
  VAR_INPUT
    RES : REAL;
    R0 : REAL;
  END_VAR

  TEMP_NI := (SQRT(0.30085225 - 2.66E-3 * (R0 - Res)) - 0.5485) * 751.8796992;

  (* From OSCAT Library, www.oscat.de *)
END_FUNCTION

FUNCTION RES_PT : REAL
  VAR_INPUT
    _T : REAL;
    R0 : REAL;
  END_VAR
  VAR
    T2 : REAL;
  END_VAR

  T2 := _T * _T;

  IF _T >= 0.0 THEN
  	RES_PT := R0 * ( 1.0 + 3.90802E-3 * _T + -5.802E-7 * T2);
  ELSE
  	RES_PT := R0 * ( 1.0 + 3.90802E-3 * _T + -5.802E-7 * T2 + -4.27350E-12 * (_T - 100.0) * T2 * _T);
  END_IF;

  (* From OSCAT Library, www.oscat.de *)
END_FUNCTION

FUNCTION TEMP_PT : REAL
  VAR_INPUT
    RES : REAL;
    R0 : REAL;
  END_VAR
  VAR
    _step : REAL := 50.0;
    X : REAL;
    Y : REAL;
    t1 : REAL;
  END_VAR

  X := 3.9083E-3 * R0;
  Y := -5.775E-7 * R0;
  IF Res >= R0 THEN
  	t1 := X * X - 4.0 * Y * (R0 - Res);
  	IF t1 < 0.0 THEN
  		TEMP_PT := 10000.0;
  	ELSE
  		TEMP_PT := (-X + SQRT(t1)) / (2.0 * Y);
  	END_IF;
  ELSE
  	(* since the formula cannot be solved this is a successive approximation *)
  	TEMP_PT := -100.0;
  	WHILE _step > 0.01 DO
  		(* test if result greater or less *)
  		IF RES_PT(TEMP_PT, R0) < res THEN TEMP_PT := TEMP_PT + _step; ELSE TEMP_PT := TEMP_PT - _step; END_IF;
  		_step := _step * 0.5;
  	END_WHILE;
  END_IF;

  (* From OSCAT Library, www.oscat.de *)
END_FUNCTION

FUNCTION MID3 : REAL
  VAR_INPUT
    IN1 : REAL;
    IN2 : REAL;
    IN3 : REAL;
  END_VAR
  VAR
    _IN1 : REAL;
    _IN2 : REAL;
    _IN3 : REAL;
  END_VAR

  _IN1 := IN1; (* VAR_INPUT auf Variablen umkopieren , da diese schreibgeschützt sind *)
  _IN2 := IN2;
  _IN3 := IN3;

  IF _IN1 > _IN2 THEN MID3 := _IN1; _IN1 := _IN2; _IN2 := MID3; END_IF;
  IF _IN2 > _IN3 THEN _IN2 := _IN3; END_IF;
  MID3 := SEL(_IN1 > _IN2, _IN2, _IN1);
  (* from OSCAT library; www.oscat.de  *)
END_FUNCTION

FUNCTION MULTI_IN : REAL
  VAR_INPUT
    IN_1 : REAL;
    IN_2 : REAL;
    IN_3 : REAL;
    DEFAULT : REAL;
    IN_MIN : REAL;
    IN_MAX : REAL;
    MODE : BYTE;
  END_VAR
  VAR
    count : INT;
    F1 : BOOL;
    F2 : BOOL;
    F3 : BOOL;
  END_VAR

  F1 :=  in_1 > in_min AND in_1 < in_max;
  F2 :=  in_2 > in_min AND in_2 < in_max;
  F3 :=  in_3 > in_min AND in_3 < in_max;

  CASE BYTE_TO_INT(mode) OF
  0:	count := 0;
  	IF F1 THEN
  		count := count + 1;
  		MULTI_IN := in_1;
  	ELSE
  		MULTI_IN := 0.0;
  	END_IF;
  	IF F2 THEN
  		count := count + 1;
  		MULTI_IN := MULTI_IN + in_2;
  	END_IF;
  	IF F3 THEN
  		count := count + 1;
  		MULTI_IN := MULTI_IN + in_3;
  	END_IF;
  	MULTI_IN := SEL(count = 0, MULTI_IN / INT_TO_REAL(count), default);

  1:	MULTI_IN := SEL(F1, default, IN_1);

  2:	MULTI_IN := SEL(F2, default, IN_2);

  3:	MULTI_IN := SEL(F3, default, IN_3);

  4:	MULTI_IN := default;

  5:	MULTI_IN := SEL(F1, in_max, IN_1);
  	IF F2 AND in_2 < MULTI_IN THEN MULTI_IN := in_2; END_IF;
  	IF F3 AND in_3 < MULTI_IN THEN MULTI_IN := in_3; END_IF;
  	IF MULTI_IN = in_max THEN MULTI_IN := default; END_IF;

  6:	MULTI_IN := SEL(F1, in_min, IN_1);
  	IF F2 AND in_2 > MULTI_IN THEN MULTI_IN := in_2; END_IF;
  	IF F3 AND in_3 > MULTI_IN THEN MULTI_IN := in_3; END_IF;
  	IF MULTI_IN = in_min THEN MULTI_IN := default; END_IF;

  7:	IF F1 AND F2 AND F3 THEN MULTI_IN := MID3(in_1, in_2, in_3);
  	ELSIF F1 AND F2 THEN MULTI_IN := MIN(in_1, in_2);
  	ELSIF F1 AND F3 THEN MULTI_IN := MIN(in_1, in_3);
  	ELSIF F2 AND F3 THEN MULTI_IN := MIN(in_2, in_3);
  	ELSIF F1 THEN MULTI_IN := in_1;
  	ELSIF F2 THEN MULTI_IN := in_2;
  	ELSIF F3 THEN MULTI_IN := in_3;
  	ELSE MULTI_IN := default;
  	END_IF;

  END_CASE;

  (* From OSCAT Library, www.oscat.de *)
  (* MID3 required *)
END_FUNCTION

PROGRAM program0
  VAR
    LocalVar0 : DINT;
    LocalVar1 : DINT;
    LocalVar2 : DINT;
    ADD1_OUT : DINT;
  END_VAR

  ADD1_OUT := ADD(LocalVar0, LocalVar1);
  LocalVar2 := ADD1_OUT;
END_PROGRAM

FUNCTION TEMP_SI : REAL
  VAR_INPUT
    RES : REAL;
    _RS : REAL;
    TS : REAL;
  END_VAR

  TEMP_SI := (-7.64E-3 + SQRT(Res/_RS* 6.64E-5 - 0.803E-5)) * 30120.48193 + TS;

  (* From OSCAT Library, www.oscat.de *)
END_FUNCTION

FUNCTION RES_NI : REAL
  VAR_INPUT
    _T : REAL;
    R0 : REAL;
  END_VAR
  VAR
    T2 : REAL;
  END_VAR

  T2 := _T*_T;
  Res_NI := R0 + 0.5485*_T + 0.665E-3*T2 + 2.805E-9*T2*T2;

  (* From OSCAT Library, www.oscat.de *)
END_FUNCTION

FUNCTION RES_NTC : REAL
  VAR_INPUT
    _T : REAL;
    RN : REAL;
    B : REAL;
  END_VAR

  RES_NTC := RN * EXP(B * (1.0 / (_T+273.15) - 0.00335401643468053));

  (* From OSCAT Library, www.oscat.de *)
END_FUNCTION

FUNCTION TEMP_NTC : REAL
  VAR_INPUT
    RES : REAL;
    RN : REAL;
    B : REAL;
  END_VAR

  IF res > 0.0 THEN
  	TEMP_NTC := B * 298.15 / (B + LN(RES / RN) * 298.15) -273.15;
  END_IF;

  (* From OSCAT Library, www.oscat.de *)
END_FUNCTION

FUNCTION SENSOR_INT : REAL
  VAR_INPUT
    VOLTAGE : REAL;
    CURRENT : REAL;
    RP : REAL;
    _RS : REAL;
  END_VAR
  VAR
    RG : REAL;
  END_VAR

  IF current <> 0.0 THEN
  	RG := voltage / current;
  	SENSOR_INT := RP * ( RG - _RS) / ( RP + _RS - RG);
  END_IF;

  (* From OSCAT Library, www.oscat.de *)
END_FUNCTION

FUNCTION RES_SI : REAL
  VAR_INPUT
    _T : REAL;
    _RS : REAL;
    TS : REAL;
  END_VAR
  VAR
    TX : REAL;
  END_VAR

  TX := _T - TS;
  RES_SI := _RS * ( 1.0 + 7.64E-3 * TX + 1.66E-5 * TX * TX);

  (* From OSCAT Library, www.oscat.de *)
END_FUNCTION

CONFIGURATION Config0

  RESOURCE Res0 ON PLC
    TASK task0(INTERVAL := T#20ms,PRIORITY := 0);
    PROGRAM instance0 WITH task0 : program0;
  END_RESOURCE
END_CONFIGURATION

(* ---- lb_claude_assisted_e6326078b5c1_0009.st ---- *)
TYPE
  LOGLEVEL : (CRITICAL, WARNING, INFO, DEBUG) := INFO;
END_TYPE

FUNCTION_BLOCK LOGGER
  VAR_INPUT
    TRIG : BOOL;
    MSG : STRING;
    LEVEL : LOGLEVEL := INFO;
  END_VAR
  VAR
    TRIG0 : BOOL;
  END_VAR

  IF TRIG AND NOT TRIG0 THEN
  {{
   LogMessage(GetFbVar(LEVEL),(char*)GetFbVar(MSG, .body),GetFbVar(MSG, .len));
  }}
  END_IF;
  TRIG0:=TRIG;
END_FUNCTION_BLOCK

PROGRAM program0
  VAR_IN_OUT
    StartButton : BOOL;
    RollerEngine : BOOL;
    Nozzle : BOOL;
    BottleSensor : BOOL;
    WaterLevelSensor : BOOL;
    PlantState : INT;
  END_VAR

  (* Initialization Phase*)
      IF PlantState = 0 THEN
          RollerEngine := FALSE;
          Nozzle := FALSE;
          IF StartButton THEN
              PlantState := 1;         (* Move to Filling Phase*)
          END_IF;
      END_IF;

      (*Filling Phase*)
      IF PlantState = 1 THEN
          IF BottleSensor AND NOT WaterLevelSensor THEN
              Nozzle := TRUE;         (*Open the nozzle if bottle is under and not filled*)
          ELSE
              Nozzle := FALSE;        (* Close the nozzle otherwise*)
          END_IF;

          IF WaterLevelSensor THEN
              PlantState := 2;        (*Move to Moving Phase once bottle is filled*)
          END_IF;
      END_IF;

      (*Moving Phase*)
      IF PlantState = 2 THEN
          Nozzle := FALSE;            (* Ensure nozzle is closed*)
          RollerEngine := TRUE;        (* Start the roller engine to move the bottle*)

          IF NOT BottleSensor THEN
              PlantState := 1;         (*Move back to Filling Phase once bottle has moved away*)
          END_IF;
      END_IF;

    (* Stop the plant if StartButton is turned off*)
      IF NOT StartButton THEN
          PlantState := 0;
      END_IF;
END_PROGRAM

CONFIGURATION Config0

  RESOURCE Res0 ON PLC
    TASK task0(INTERVAL := T#20ms,PRIORITY := 0);
    PROGRAM instance0 WITH task0 : program0;
  END_RESOURCE
END_CONFIGURATION

(* ---- lb_claude_assisted_e9068fe2c077_0079.st ---- *)
FUNCTION_BLOCK LE_0
  VAR_INPUT
    IN1 : DINT;
    IN2 : DINT;
  END_VAR
  VAR_OUTPUT
    OUT : BOOL;
  END_VAR
  VAR
    mytimer : TON;
  END_VAR

  OUT:=FALSE;
  IF IN1<=IN2 then
    OUT:=TRUE;
  END_IF;
  mytimer(IN := TRUE, PT := t#8000ms);

  IF mytimer.Q = TRUE then

      OUT:=TRUE;

  End_IF;
END_FUNCTION_BLOCK

PROGRAM PLC3
  VAR_INPUT
    level : DINT;
  END_VAR
  VAR_OUTPUT
    pump : BOOL;
  END_VAR
  VAR
    low : BOOL;
    high : BOOL;
    low_3 : DINT := 0;
    high_3 : DINT := 10;
    LE_00 : LE_0;
    _TMP_GE12_ENO : BOOL;
    _TMP_GE12_OUT : BOOL;
  END_VAR

  _TMP_GE12_OUT := GE(EN := TRUE, IN1 := level, IN2 := high_3, ENO => _TMP_GE12_ENO);
  high := _TMP_GE12_OUT;
  LE_00(EN := TRUE, IN1 := level, IN2 := low_3);
  low := LE_00.OUT;
  pump := NOT(low) AND (high OR pump);
END_PROGRAM

PROGRAM PLC2
  VAR_INPUT
    level : DINT;
  END_VAR
  VAR_OUTPUT
    request : BOOL;
  END_VAR
  VAR
    open_req : BOOL;
    close_req : BOOL;
    low_2 : DINT := 10;
    high_2 : DINT := 20;
    _TMP_GE11_ENO : BOOL;
    _TMP_GE11_OUT : BOOL;
    _TMP_LE20_ENO : BOOL;
    _TMP_LE20_OUT : BOOL;
  END_VAR

  _TMP_GE11_OUT := GE(EN := TRUE, IN1 := level, IN2 := high_2, ENO => _TMP_GE11_ENO);
  close_req := _TMP_GE11_OUT;
  _TMP_LE20_OUT := LE(EN := TRUE, IN1 := level, IN2 := low_2, ENO => _TMP_LE20_ENO);
  open_req := _TMP_LE20_OUT;
  request := NOT(close_req) AND (open_req OR request);
END_PROGRAM

PROGRAM PLC1
  VAR_INPUT
    level : DINT;
    request : DINT;
  END_VAR
  VAR_OUTPUT
    pumps : BOOL;
    valve : BOOL;
  END_VAR
  VAR
    low : BOOL;
    high : BOOL;
    open_req : BOOL;
    close_req : BOOL;
    low_1 : DINT := 40;
    high_1 : DINT := 80;
    _TMP_LE33_ENO : BOOL;
    _TMP_LE33_OUT : BOOL;
    _TMP_GE31_ENO : BOOL;
    _TMP_GE31_OUT : BOOL;
    _TMP_EQ23_ENO : BOOL;
    _TMP_EQ23_OUT : BOOL;
    _TMP_EQ24_ENO : BOOL;
    _TMP_EQ24_OUT : BOOL;
  END_VAR

  _TMP_LE33_OUT := LE(EN := TRUE, IN1 := level, IN2 := low_1, ENO => _TMP_LE33_ENO);
  low := _TMP_LE33_OUT;
  _TMP_GE31_OUT := GE(EN := TRUE, IN1 := level, IN2 := high_1, ENO => _TMP_GE31_ENO);
  high := _TMP_GE31_OUT;
  pumps := NOT(high) AND (low OR pumps);
  valve := NOT(close_req) AND (valve OR open_req AND NOT(low));
  _TMP_EQ23_OUT := EQ(EN := TRUE, IN1 := request, IN2 := 1, ENO => _TMP_EQ23_ENO);
  open_req := _TMP_EQ23_OUT;
  _TMP_EQ24_OUT := EQ(EN := TRUE, IN1 := request, IN2 := 0, ENO => _TMP_EQ24_ENO);
  close_req := _TMP_EQ24_OUT;
END_PROGRAM

CONFIGURATION Config0

  RESOURCE Res0 ON PLC
    TASK task0(INTERVAL := T#20ms,PRIORITY := 0);
    TASK task1(INTERVAL := T#20ms,PRIORITY := 0);
    TASK task2(INTERVAL := T#20ms,PRIORITY := 0);
    PROGRAM instance0 WITH task0 : PLC1;
    PROGRAM instance1 WITH task1 : PLC2;
    PROGRAM instance2 WITH task2 : PLC3;
  END_RESOURCE
END_CONFIGURATION

(* ---- lb_claude_assisted_e95623b0af83_0052.st ---- *)
FUNCTION_BLOCK T_PLC_US_Block

	VAR_OUTPUT
		T_PLC_US :	UDINT;
	END_VAR

	VAR_EXTERNAL
		PLC_TICKS_PER_SEC :	INT;
		PLC_SYS_TICK_CNT :	DINT;
	END_VAR

	VAR
		debug :	BOOL;
		N :	INT;
		Offset :	UDINT;
		temp :	DWORD := DWORD#1;
		mode :	BOOL;
		faktor :	UDINT;
		init :	BOOL;
		v_plc_ticks_per_sec :	UDINT;
		base :	UDINT := UDINT#1000000;
	END_VAR

	IF init = FALSE THEN
		v_plc_ticks_per_sec := INT_TO_UDINT(PLC_TICKS_PER_SEC);
		IF v_plc_ticks_per_sec = UDINT#1024 THEN
			faktor := UDINT#1000;
			mode := FALSE;
		ELSIF v_plc_ticks_per_sec > UDINT#0 THEN
			IF v_plc_ticks_per_sec <= base THEN
				faktor := base / v_plc_ticks_per_sec;
				mode := FALSE;
			ELSE
				faktor := v_plc_ticks_per_sec / base;
				mode := TRUE;
			END_IF;
		ELSE
			faktor := UDINT#1;
		END_IF;
		init := TRUE;
	END_IF;

	IF mode THEN
		T_PLC_US := DINT_TO_UDINT(PLC_SYS_TICK_CNT) / faktor;
	ELSE
		T_PLC_US := DINT_TO_UDINT(PLC_SYS_TICK_CNT) * faktor;
	END_IF;

	IF debug THEN
		T_PLC_US := (DWORD_TO_UDINT(SHL(UDINT_TO_DWORD(T_PLC_US),N) OR SHL(temp,N)) - UDINT#1) + Offset;
	END_IF;
END_FUNCTION_BLOCK

FUNCTION_BLOCK FT_PT1

	VAR_INPUT
		IN :	REAL;
		T :	TIME;
		K :	REAL := 1.0;
	END_VAR

	VAR_OUTPUT
		OUT :	REAL;
	END_VAR

	VAR
		last :	UDINT;
		tx :	UDINT;
		init :	BOOL;
		T_PLC_US :	T_PLC_US_Block;
	END_VAR

	T_PLC_US();
	tx:= T_PLC_US.T_PLC_US;

	IF NOT init OR T = t#0s THEN
		init := TRUE;
		out := K * in;
	ELSE
		out := out + (in * K - out) * UDINT_TO_REAL(Tx - last) / TIME_TO_REAL(T) * 1.0E-3;
		IF ABS(out) < 1.0E-20 THEN out := 0.0; END_IF;
	END_IF;
	last := tx;
END_FUNCTION_BLOCK

FUNCTION _REAL_TO_DWORD: DWORD

  VAR_INPUT
    X :	REAL;
  END_VAR

  IF REAL_TO_DWORD(0.5) = DWORD#1 THEN
    _REAL_TO_DWORD := REAL_TO_DWORD(x);
  ELSIF X > 0.0 THEN
    _REAL_TO_DWORD := REAL_TO_DWORD(x+0.5);
  ELSIF X < 0.0 THEN
    _REAL_TO_DWORD := REAL_TO_DWORD(x-0.5);
  ELSE
    _REAL_TO_DWORD := DWORD#0;
  END_IF;
END_FUNCTION

FUNCTION _DWORD_TO_REAL:REAL
	VAR_INPUT
		IN :	DWORD;
	END_VAR

	_DWORD_TO_REAL := UDINT_TO_REAL(DWORD_TO_UDINT(IN));
END_FUNCTION

FUNCTION MULTIME:TIME
	VAR_INPUT
		T :	TIME;
		M :	REAL;
	END_VAR

	multime := DWORD_TO_TIME(_REAL_TO_DWORD(_DWORD_TO_REAL(TIME_TO_DWORD(t))*M));
END_FUNCTION

FUNCTION_BLOCK DEAD_BAND_A
	VAR_INPUT
		X :	REAL;
		T :	TIME;
		KL :	REAL := 1.0;
		LM :	REAL;
	END_VAR

	VAR_OUTPUT
		Y :	REAL;
		L :	REAL;
	END_VAR

	VAR
		tp1 :	FT_PT1;
		tp2 :	FT_PT1;
	END_VAR

	tp1(in := X, T:= T);
	tp2(in := ABS(tp1.out - X), T := MULTIME(T, 4.0));
	L := MIN(KL * tp2.out, LM);

	IF X > L THEN
		Y := X - L;
	ELSIF X < -L THEN
		Y := X + L;
	ELSE
		Y := 0.0;
	END_IF;
END_FUNCTION_BLOCK

PROGRAM program0
  VAR

		X  :	REAL;
		T  :	TIME;
		KL :	REAL;
		LM :	REAL;

		Y :	REAL;
		L :	REAL;

	func_block : DEAD_BAND_A;
  END_VAR
	func_block.X   :=X ;
	func_block.T   :=T ;
	func_block.KL  :=KL;
	func_block.LM  :=LM;
	func_block();
	Y := func_block.Y;
	L := func_block.L;
END_PROGRAM

CONFIGURATION Config0

	VAR_GLOBAL
		PLC_TICKS_PER_SEC :	INT;
		PLC_SYS_TICK_CNT :	DINT;
	END_VAR

	RESOURCE Res0 ON PLC
		TASK task0(INTERVAL := T#20ms,PRIORITY := 0);
		PROGRAM instance0 WITH task0 : program0;
	END_RESOURCE

END_CONFIGURATION

(* ---- lb_claude_assisted_eb47d59fc93f_0004.st ---- *)
(*
This code implements a randomly grown symbolic expression:

(xor(xor(IN40, IN23), IN33)) | IN36

*)

FUNCTION_BLOCK F_CollectInput
  VAR_IN_OUT
      Data : ARRAY[1..50] OF BOOL;
  END_VAR
  VAR_INPUT
      TICK  : BOOL := 0;
      IN1   : BOOL := 0;
      IN2   : BOOL := 0;
      IN3   : BOOL := 0;
      IN4   : BOOL := 0;
      IN5   : BOOL := 0;
      RESET : BOOL := FALSE;
  END_VAR
  VAR_OUTPUT
      Finished : BOOL;
  END_VAR
  VAR
      j    : USINT := 1;
      tock : BOOL  := 0;
  END_VAR
  IF NOT RESET AND tock = NOT TICK THEN
      Data[j]   := IN1;
      Data[j+1] := IN2;
      Data[j+2] := IN3;
      Data[j+3] := IN4;
      Data[j+4] := IN5;
      j := j + 5;
      tock := TICK;
  ELSE
      j := 1;
      tock := 0;
  END_IF;
  Finished := (j > 50);
END_FUNCTION_BLOCK

PROGRAM Boiler
  VAR
    Data  : ARRAY[1..50] OF BOOL;
    Ready : BOOL;
    CollectInput : F_CollectInput;
  END_VAR
  VAR
    TICK     AT %IX1.0 : BOOL;
    IN1      AT %IX0.3 : BOOL;
    IN2      AT %IX0.4 : BOOL;
    IN3      AT %IX0.5 : BOOL;
    IN4      AT %IX0.6 : BOOL;
    IN5      AT %IX0.7 : BOOL;
    OutReady AT %QX0.0 : BOOL := FALSE;
    FeedNext AT %QX0.1 : BOOL := FALSE;
    Out      AT %QX0.2 : BOOL;
  END_VAR
  CollectInput(TICK:=TICK, IN1:=IN1, IN2:=IN2, IN3:=IN3, IN4:=IN4, IN5:=IN5);
  Ready := CollectInput.Finished;
  FeedNext := 1;
  IF Ready THEN
    Out := (((Data[40] XOR Data[23]) XOR Data[33]) OR Data[36]);
    OutReady := 1;
    CollectInput(RESET:=TRUE);
  END_IF;
END_PROGRAM

CONFIGURATION Config0
  RESOURCE Res0 ON PLC
    TASK task0(INTERVAL := T#20ms,PRIORITY := 0);
    PROGRAM instance0 WITH task0 : Boiler;
  END_RESOURCE
END_CONFIGURATION

(* ---- lb_claude_assisted_ec691a330eba_0011.st ---- *)
FUNCTION UDINT_TO_TIME2:TIME

	VAR_INPUT
		IN :	UDINT;
	END_VAR

	UDINT_TO_TIME2 := DINT_TO_TIME(UDINT_TO_DINT(IN));

END_FUNCTION

FUNCTION_BLOCK T_PLC_MS_block
	VAR_OUTPUT
		T_PLC_MS :	UDINT;
	END_VAR

	VAR_EXTERNAL
		PLC_TICKS_PER_SEC :	INT;
		PLC_SYS_TICK_CNT :	DINT;
	END_VAR

	VAR
		debug :	BOOL;(*Debug-Mode ON / OFF*)
		N :	INT;(*Debug-Faktor*)
		Offset :	UDINT;(*Debug-Offset*)
		temp :	DWORD := DWORD#1;(*Debug-Offset*)
		mode :	BOOL;(*modus*)
		faktor :	UDINT;(*Systemtakt-Faktor*)
		init :	BOOL;
		v_plc_ticks_per_sec :	UDINT;
		base :	UDINT := UDINT#1000;
	END_VAR

	IF init = FALSE THEN
		v_plc_ticks_per_sec := INT_TO_UDINT(PLC_TICKS_PER_SEC);
		IF v_plc_ticks_per_sec = UDINT#1024 THEN
			faktor := UDINT#1;
			mode := FALSE;
		ELSIF v_plc_ticks_per_sec > UDINT#0 THEN
			IF v_plc_ticks_per_sec <= base THEN
				faktor := base / v_plc_ticks_per_sec;
				mode := FALSE;
			ELSE
				faktor := v_plc_ticks_per_sec / base;
				mode := TRUE;
			END_IF;
		ELSE
			faktor := UDINT#1;
		END_IF;
		init := TRUE;
	END_IF;

	IF mode THEN
		T_PLC_MS := DINT_TO_UDINT(PLC_SYS_TICK_CNT) / faktor;
	ELSE
		T_PLC_MS := DINT_TO_UDINT(PLC_SYS_TICK_CNT) * faktor;
	END_IF;

	IF debug THEN
		T_PLC_MS := (DWORD_TO_UDINT(SHL(UDINT_TO_DWORD(T_PLC_MS),N) OR SHL(temp,N)) - UDINT#1) + Offset;
	END_IF;

END_FUNCTION_BLOCK

FUNCTION TIME_TO_UDINT2:UDINT
	VAR_INPUT
		X :	TIME;
	END_VAR

	TIME_TO_UDINT2 := DINT_TO_UDINT(TIME_TO_DINT(X));
END_FUNCTION

FUNCTION FRMP_B:BYTE
	VAR_INPUT
		START :	BYTE;
		DIR :	BOOL;
		TD :	TIME;
		TR :	TIME;
	END_VAR

	IF TD < TR THEN
		FRMP_B := MIN(UDINT_TO_BYTE(DWORD_TO_UDINT(SHL(TIME_TO_DWORD(TD), 8)) / TIME_TO_UDINT2(TR)), SEL(DIR, START, USINT_TO_BYTE(USINT#255 - BYTE_TO_USINT(START))));
		IF DIR THEN
			FRMP_B := USINT_TO_BYTE(BYTE_TO_USINT(START) + BYTE_TO_USINT(FRMP_B));
		ELSE
			FRMP_B := USINT_TO_BYTE(BYTE_TO_USINT(START) - BYTE_TO_USINT(FRMP_B));
		END_IF;
	ELSE
		FRMP_B := SEL(DIR, BYTE#0, BYTE#255);
	END_IF;
END_FUNCTION

FUNCTION_BLOCK _RMP_B
	VAR_INPUT
		DIR :	BOOL;
		E :	BOOL := TRUE;
		TR :	TIME;
	END_VAR

	VAR_IN_OUT
		RMP :	BYTE;
	END_VAR

	VAR
		T_PLC_MS :	T_PLC_MS_block;
		tx :	TIME;
		tl :	TIME;
		tn :	TIME;
		init :	BOOL;
		last_dir :	BOOL;
		start :	BYTE;
	END_VAR

	T_PLC_MS();
	tx := UDINT_TO_TIME(T_PLC_MS.T_PLC_MS);

	IF E AND init AND (dir = last_dir) AND (RMP <> SEL(DIR, BYTE#0, BYTE#255)) AND TR = tn THEN
		RMP := FRMP_B(start, DIR, tx - tl, TR);
	ELSE
		init := TRUE;
		tl := tx;
		tn := tr;
		start := RMP;
	END_IF;
	last_dir := dir;
END_FUNCTION_BLOCK

FUNCTION_BLOCK AUTORUN_Block

	VAR_INPUT
		IN :	BOOL;
		TEST :	BOOL;
		ARE :	BOOL := TRUE;
		TRUN :	TIME;
		TOFF :	TIME;
	END_VAR

	VAR_OUTPUT
		OUT :	BOOL;
		ARO :	BOOL;
	END_VAR

	VAR_IN_OUT
		ARX :	BOOL;
	END_VAR

	VAR
		timer :	_RMP_B;
		val :	BYTE;
	END_VAR

	IF TOFF > T#0s THEN
		timer(DIR:= OUT, TR := SEL(OUT, TOFF, TRUN), RMP := val);
		val := timer.RMP;
	ELSE
		val := BYTE#255;
	END_IF;

	IF (NOT ARX AND ARE AND val = BYTE#0) OR TEST THEN
		val := BYTE#0;
		ARO := TRUE;
		ARX := TRUE;
	ELSIF val = BYTE#255 AND ARO THEN
		ARO := FALSE;
		ARX := FALSE;
	END_IF;

	out := IN OR ARO;

END_FUNCTION_BLOCK

PROGRAM program0
	VAR
		IN :	BOOL;
		TEST :	BOOL;
		ARE :	BOOL := TRUE;
		TRUN :	TIME;
		TOFF :	TIME;
		OUT :	BOOL;
		ARO :	BOOL;
		func_block : AUTORUN_Block;
	END_VAR
	func_block.IN := IN;
	func_block.TEST := TEST;
	func_block.ARE := ARE ;
	func_block.TRUN := TRUN;
	func_block.TOFF := TOFF;
	func_block();
	OUT  := func_block.OUT;
	ARO  := func_block.ARO;
END_PROGRAM

CONFIGURATION Config0
	VAR_GLOBAL
		PLC_TICKS_PER_SEC :	INT;
		PLC_SYS_TICK_CNT :	DINT;
	END_VAR
  	RESOURCE Res0 ON PLC
    	TASK task0(INTERVAL := T#20ms,PRIORITY := 0);
    	PROGRAM instance0 WITH task0 : program0;
  	END_RESOURCE
END_CONFIGURATION

(* ---- lb_claude_assisted_ee197bfeae12_0067.st ---- *)
TYPE
  LOGLEVEL : (CRITICAL, WARNING, INFO, DEBUG) := INFO;
END_TYPE

FUNCTION_BLOCK LOGGER
  VAR_INPUT
    TRIG : BOOL;
    MSG : STRING;
    LEVEL : LOGLEVEL := INFO;
  END_VAR
  VAR
    TRIG0 : BOOL;
  END_VAR

  IF TRIG AND NOT TRIG0 THEN
  {{
   LogMessage(GetFbVar(LEVEL),(char*)GetFbVar(MSG, .body),GetFbVar(MSG, .len));
  }}
  END_IF;
  TRIG0:=TRIG;
END_FUNCTION_BLOCK

FUNCTION_BLOCK python_eval
  VAR_INPUT
    TRIG : BOOL;
    CODE : STRING;
  END_VAR
  VAR_OUTPUT
    ACK : BOOL;
    RESULT : STRING;
  END_VAR
  VAR
    STATE : DWORD;
    BUFFER : STRING;
    PREBUFFER : STRING;
    TRIGM1 : BOOL;
    TRIGGED : BOOL;
  END_VAR

  {extern void __PythonEvalFB(int, PYTHON_EVAL*);__PythonEvalFB(0, data__);}
END_FUNCTION_BLOCK

FUNCTION_BLOCK python_poll
  VAR_INPUT
    TRIG : BOOL;
    CODE : STRING;
  END_VAR
  VAR_OUTPUT
    ACK : BOOL;
    RESULT : STRING;
  END_VAR
  VAR
    STATE : DWORD;
    BUFFER : STRING;
    PREBUFFER : STRING;
    TRIGM1 : BOOL;
    TRIGGED : BOOL;
  END_VAR

  {extern void __PythonEvalFB(int, PYTHON_EVAL*);__PythonEvalFB(1,(PYTHON_EVAL*)(void*)data__);}
END_FUNCTION_BLOCK

FUNCTION_BLOCK python_gear
  VAR_INPUT
    N : UINT;
    TRIG : BOOL;
    CODE : STRING;
  END_VAR
  VAR_OUTPUT
    ACK : BOOL;
    RESULT : STRING;
  END_VAR
  VAR
    py_eval : python_eval;
    COUNTER : UINT;
    ADD10_OUT : UINT;
    EQ13_OUT : BOOL;
    SEL15_OUT : UINT;
    AND7_OUT : BOOL;
  END_VAR

  ADD10_OUT := ADD(COUNTER, 1);
  EQ13_OUT := EQ(N, ADD10_OUT);
  SEL15_OUT := SEL(EQ13_OUT, ADD10_OUT, 0);
  COUNTER := SEL15_OUT;
  AND7_OUT := AND(EQ13_OUT, TRIG);
  py_eval(TRIG := AND7_OUT, CODE := CODE);
  ACK := py_eval.ACK;
  RESULT := py_eval.RESULT;
END_FUNCTION_BLOCK

PROGRAM part1c
  VAR
    Input0 : BOOL;
    Output0 : BOOL;
  END_VAR
  VAR
    Oscillator : BOOL;
    TON0 : TON;
    TOF0 : TOF;
    CTU0 : CTU;
    Bomb : BOOL;
    Countup : INT := 5;
    TrueBool : BOOL := 1;
    TON1 : TON;
    R_TRIG1 : R_TRIG;
  END_VAR

  TON0(IN := NOT(Oscillator) AND Input0, PT := T#6000ms);
  TOF0(IN := TON0.Q, PT := T#6000ms);
  Oscillator := TOF0.Q;
  Output0 := NOT(Oscillator) AND Input0 OR Bomb;
  R_TRIG1(CLK := Output0);
  CTU0(CU := R_TRIG1.Q, PV := Countup);
  TON1(IN := Input0, PT := T#30000ms);
  Bomb := Bomb OR CTU0.Q OR TON1.Q;
END_PROGRAM

CONFIGURATION Config0

  RESOURCE Res0 ON PLC
    TASK task0(INTERVAL := T#20ms,PRIORITY := 0);
    PROGRAM instance0 WITH task0 : part1c;
  END_RESOURCE
END_CONFIGURATION

(* ---- lb_claude_assisted_ee3fe1ae7f79_0015.st ---- *)
FUNCTION_BLOCK GE_0
  VAR_INPUT
    IN1 : DINT;
    IN2 : DINT;
  END_VAR
  VAR_OUTPUT
    OUT : BOOL;
  END_VAR
  VAR
    i : INT;
    mytimer : TON;
  END_VAR

  OUT:=FALSE;
  IF IN1>=IN2 then
    OUT:=TRUE;
  END_IF;

  mytimer(IN := TRUE, PT := t#8000ms);
  i:=0;
  IF mytimer.Q = TRUE then
     WHILE i<4 do
      OUT:=TRUE;
    End_WHILE;
  End_IF;
END_FUNCTION_BLOCK

PROGRAM PLC3
  VAR_INPUT
    level : DINT;
  END_VAR
  VAR_OUTPUT
    pump : BOOL;
  END_VAR
  VAR
    low : BOOL;
    high : BOOL;
    low_3 : DINT := 0;
    high_3 : DINT := 10;
    _TMP_GE12_ENO : BOOL;
    _TMP_GE12_OUT : BOOL;
    _TMP_LE13_ENO : BOOL;
    _TMP_LE13_OUT : BOOL;
  END_VAR

  _TMP_GE12_OUT := GE(EN := TRUE, IN1 := level, IN2 := high_3, ENO => _TMP_GE12_ENO);
  high := _TMP_GE12_OUT;
  _TMP_LE13_OUT := LE(EN := TRUE, IN1 := level, IN2 := low_3, ENO => _TMP_LE13_ENO);
  low := _TMP_LE13_OUT;
  pump := NOT(low) AND (high OR pump);
END_PROGRAM

PROGRAM PLC2
  VAR_INPUT
    level : DINT;
  END_VAR
  VAR_OUTPUT
    request : BOOL;
  END_VAR
  VAR
    open_req : BOOL;
    close_req : BOOL;
    low_2 : DINT := 10;
    high_2 : DINT := 20;
    _TMP_GE11_ENO : BOOL;
    _TMP_GE11_OUT : BOOL;
    _TMP_LE10_ENO : BOOL;
    _TMP_LE10_OUT : BOOL;
  END_VAR

  _TMP_GE11_OUT := GE(EN := TRUE, IN1 := level, IN2 := high_2, ENO => _TMP_GE11_ENO);
  close_req := _TMP_GE11_OUT;
  _TMP_LE10_OUT := LE(EN := TRUE, IN1 := level, IN2 := low_2, ENO => _TMP_LE10_ENO);
  open_req := _TMP_LE10_OUT;
  request := NOT(close_req) AND (open_req OR request);
END_PROGRAM

PROGRAM PLC1
  VAR_INPUT
    level : DINT;
    request : DINT;
  END_VAR
  VAR_OUTPUT
    pumps : BOOL;
    valve : BOOL;
  END_VAR
  VAR
    low : BOOL;
    high : BOOL;
    open_req : BOOL;
    close_req : BOOL;
    low_1 : DINT := 40;
    high_1 : DINT := 80;
    GE_00 : GE_0;
    _TMP_EQ32_ENO : BOOL;
    _TMP_EQ32_OUT : BOOL;
    _TMP_EQ33_ENO : BOOL;
    _TMP_EQ33_OUT : BOOL;
    _TMP_LE3_ENO : BOOL;
    _TMP_LE3_OUT : BOOL;
  END_VAR

  _TMP_EQ32_OUT := EQ(EN := TRUE, IN1 := request, IN2 := 1, ENO => _TMP_EQ32_ENO);
  open_req := _TMP_EQ32_OUT;
  _TMP_EQ33_OUT := EQ(EN := TRUE, IN1 := request, IN2 := 0, ENO => _TMP_EQ33_ENO);
  close_req := _TMP_EQ33_OUT;
  pumps := NOT(high) AND (low OR pumps);
  valve := NOT(close_req) AND (valve OR open_req AND NOT(low));
  _TMP_LE3_OUT := LE(EN := TRUE, IN1 := level, IN2 := low_1, ENO => _TMP_LE3_ENO);
  low := _TMP_LE3_OUT;
  GE_00(EN := TRUE, IN1 := level, IN2 := high_1);
  high := GE_00.OUT;
END_PROGRAM

CONFIGURATION Config0

  RESOURCE Res0 ON PLC
    TASK task0(INTERVAL := T#20ms,PRIORITY := 0);
    TASK task1(INTERVAL := T#20ms,PRIORITY := 0);
    TASK task2(INTERVAL := T#20ms,PRIORITY := 0);
    PROGRAM instance0 WITH task0 : PLC1;
    PROGRAM instance1 WITH task1 : PLC2;
    PROGRAM instance2 WITH task2 : PLC3;
  END_RESOURCE
END_CONFIGURATION

(* ---- lb_claude_assisted_eeee4f3e8ce4_0035.st ---- *)
FUNCTION_BLOCK T_PLC_MS_block
	VAR_OUTPUT
		T_PLC_MS :	UDINT;
	END_VAR

	VAR
		PLC_TICKS_PER_SEC :	INT;
		PLC_SYS_TICK_CNT :	DINT;
	END_VAR

	VAR
		debug :	BOOL;(*Debug-Mode ON / OFF*)
		N :	INT;(*Debug-Faktor*)
		Offset :	UDINT;(*Debug-Offset*)
		temp :	DWORD := DWORD#1;(*Debug-Offset*)
		MODE :	BOOL;(*modus*)
		faktor :	UDINT;(*Systemtakt-Faktor*)
		init :	BOOL;
		v_plc_ticks_per_sec :	UDINT;
		base :	UDINT := UDINT#1000;
	END_VAR

	IF init = FALSE THEN
		v_plc_ticks_per_sec := INT_TO_UDINT(PLC_TICKS_PER_SEC);
		IF v_plc_ticks_per_sec = UDINT#1024 THEN
			faktor := UDINT#1;
			MODE := FALSE;
		ELSIF v_plc_ticks_per_sec > UDINT#0 THEN
			IF v_plc_ticks_per_sec <= base THEN
				faktor := base / v_plc_ticks_per_sec;
				MODE := FALSE;
			ELSE
				faktor := v_plc_ticks_per_sec / base;
				MODE := TRUE;
			END_IF;
		ELSE
			faktor := UDINT#1;
		END_IF;
		init := TRUE;
	END_IF;

	IF MODE THEN
		T_PLC_MS := DINT_TO_UDINT(PLC_SYS_TICK_CNT) / faktor;
	ELSE
		T_PLC_MS := DINT_TO_UDINT(PLC_SYS_TICK_CNT) * faktor;
	END_IF;

	IF debug THEN
		T_PLC_MS := (DWORD_TO_UDINT(SHL(UDINT_TO_DWORD(T_PLC_MS),N) OR SHL(temp,N)) - UDINT#1) + Offset;
	END_IF;
END_FUNCTION_BLOCK

FUNCTION _WORD_TO_DINT:DINT
	VAR_INPUT
		IN :	WORD;
	END_VAR
	_WORD_TO_DINT := UINT_TO_DINT(WORD_TO_UINT(IN));
END_FUNCTION

FUNCTION TIME_TO_UDINT2:UDINT
	VAR_INPUT
		X :	TIME;
	END_VAR

	TIME_TO_UDINT2 := DINT_TO_UDINT(TIME_TO_DINT(X));
END_FUNCTION

FUNCTION_BLOCK _RMP_W

	VAR_INPUT
		DIR :	BOOL;
		E :	BOOL := TRUE;
		TR :	TIME;
	END_VAR

	VAR_IN_OUT
		RMP :	WORD;
	END_VAR

	VAR
		T_PLC_MS :	T_PLC_MS_block;
		TX :	UDINT;
		TL :	UDINT;
		PTesss :	DINT;
		init :	BOOL;
		last_DIR :	BOOL;
	END_VAR

	T_PLC_MS();
	TX := T_PLC_MS.T_PLC_MS;
	IF E AND init THEN
		(* we need to set TL = TX when DIRection CHAnges *)
		IF DIR XOR last_DIR THEN
			TL := TX;
			last_DIR := DIR;
		END_IF;
		(* check_elapsed time and calculate only if necessary *)
		IF TR > t#0s THEN
			PTesss := DWORD_TO_DINT(UDINT_TO_DWORD(DWORD_TO_UDINT(SHL(UDINT_TO_DWORD(TX- TL), 16)) / TIME_TO_UDINT2(TR)));
		ELSE
			PTesss := DINT#65535;
		END_IF;
		IF PTesss > DINT#0 THEN
			(* perform the PTesss on the ramp *)
			TL := TX;
			(* calculate the PTesss response *)
			IF NOT DIR THEN PTesss := - PTesss; END_IF;
			rmp := DINT_TO_WORD(LIMIT(DINT#0, _WORD_TO_DINT(rmp) + PTesss, DINT#65535));
		END_IF;
	ELSE
		TL := TX;
		init := TRUE;
	END_IF;
END_FUNCTION_BLOCK

FUNCTION_BLOCK RMP_W

	VAR_INPUT
		SET :	BOOL;
		PT :	TIME;
		E :	BOOL := TRUE;
		UP :	BOOL := TRUE;
		RST :	BOOL;
	END_VAR

	VAR_OUTPUT
		OUT :	WORD;
		BUSY :	BOOL;
		HIGH :	BOOL;
		LOW :	BOOL;
	END_VAR

	VAR
		rmp :	_RMP_W;
	END_VAR

	rmp(DIR := UP, E := E, TR := PT, rmp := OUT);
	OUT := rmp.RMP;

	IF RST THEN
		OUT := WORD#0;
	ELSIF SET THEN
		OUT := WORD#65535;
	END_IF;

	LOW := OUT = WORD#0;
	HIGH := OUT = WORD#65535;
	busy := NOT (low OR high) AND E;

END_FUNCTION_BLOCK

PROGRAM program0
  VAR
		SET :	BOOL;
		PT  :	TIME;
		E   :	BOOL;
		UP  :	BOOL ;
		RST :	BOOL;

		OUT  :	WORD;
		BUSY :	BOOL;
		HIGH :	BOOL;
		LOW  :	BOOL;

	func_block : RMP_W;
  END_VAR
	func_block.SET:=SET;
	func_block.PT :=PT ;
	func_block.E  :=E ;
	func_block.UP :=UP ;
	func_block.RST:=RST;
	func_block();
	OUT  := func_block.OUT ;
	BUSY := func_block.BUSY;
	HIGH := func_block.HIGH;
	LOW  := func_block.LOW ;

END_PROGRAM

(* ---- lb_claude_assisted_f22c352f1404_0055.st ---- *)
TYPE
  bya_TN_CHAR:       	ARRAY [0..1919] OF BYTE;
  bya_TN_BACKUP:     	ARRAY [0..1919] OF BYTE;
  bya_TN_COLOR:      	ARRAY [0..1919] OF BYTE;
  bya_TN_Line_Update:	ARRAY [0..23]   OF BOOL;

  us_TN_SCREEN :
  STRUCT
		bya_CHAR:			bya_TN_CHAR;
		bya_COLOR:			bya_TN_COLOR;
		bya_BACKUP:			bya_TN_BACKUP;
		bya_Line_Update:	bya_TN_Line_Update;

		by_Input_Exten_Code:    BYTE;
		by_Input_ASCII_Code:    BYTE;
		bo_Input_ASCII_IsNum:   BOOL;
		in_Page_Number:        	INT;                (* aktive Seiten-Nr.              *)
		in_Cursor_X:           	INT;                (* Cursor X-POSition              *)
		in_Cursor_Y:           	INT;                (* Cursor Y-POSition              *)
		in_EOS_Offset:         	INT;                (* End of String Offset           *)
		by_Clear_Screen_Attr:  	BYTE;               (* Clear-Screen Attr              *)
		bo_Clear_Screen:       	BOOL;               (* Clear-Screen ausl�sen          *)
		bo_Modal_Dialog:       	BOOL;               (* Modaler Dialog ist aktiv       *)
		bo_Menue_Bar_Dialog:   	BOOL;               (* Menue Dialog ist aktiv         *)

  END_STRUCT;
END_TYPE

FUNCTION TN_SC_XY2_ERROR:BOOL

	VAR_INPUT
		X1 :	INT;
		Y1 :	INT;
		X2 :	INT;
		Y2 :	INT;
	END_VAR

	TN_SC_XY2_ERROR := Y1 < 0 OR X1 < 0 OR Y2 < 0 OR X2 < 0 OR Y1 > 23 OR X1 > 79 OR Y2 > 23 OR X2 > 79;

END_FUNCTION

FUNCTION_BLOCK TN_SC_FILL_Block

	VAR
		in_X :	INT;
		in_Y :	INT;
		in_Offset :	INT;
	END_VAR

	VAR_INPUT
		Iin_Y1 :	INT;
		Iin_X1 :	INT;
		Iin_Y2 :	INT;
		Iin_X2 :	INT;
		Iby_CHAR :	BYTE;
		Iby_Attr :	BYTE;
	END_VAR

	VAR_IN_OUT
		Xus_TN_SCREEN :	us_TN_SCREEN;
	END_VAR

	IF TN_SC_XY2_ERROR(Iin_X1,Iin_Y1,Iin_X2,Iin_Y2) THEN RETURN; END_IF;

	FOR in_Y := Iin_Y1 TO Iin_Y2 DO
	Xus_TN_SCREEN.bya_Line_Update[in_Y] := TRUE;
	in_Offset := (in_Y * 80) + Iin_X1;
	FOR in_X := Iin_X1 TO Iin_X2 DO
		Xus_TN_SCREEN.bya_CHAR[in_Offset]  := Iby_CHAR;
		Xus_TN_SCREEN.bya_COLOR[in_Offset] := Iby_Attr;
		in_Offset := in_Offset + 1;
	END_FOR;
	END_FOR;

END_FUNCTION_BLOCK

FUNCTION_BLOCK TN_SC_BOX_Block

  VAR
    FB_TN_SC_FILL :	TN_SC_FILL_Block;
  END_VAR

  VAR
    by_BorderCHAR_L_T :	BYTE;
    by_BorderCHAR_T :	BYTE;
    by_BorderCHAR_B :	BYTE;
    by_BorderCHAR_R_T :	BYTE;
    by_BorderCHAR_L :	BYTE;
    by_BorderCHAR_R :	BYTE;
    by_BorderCHAR_L_B :	BYTE;
    by_BorderCHAR_R_B :	BYTE;
    in_Y :	INT;
    in_X :	INT;
    in_Border_Offset :	INT;
    in_Offset_1 :	INT;
    in_Offset_2 :	INT;
  END_VAR

  VAR_INPUT
    Iin_Y1 :	INT;
    Iin_X1 :	INT;
    Iin_Y2 :	INT;
    Iin_X2 :	INT;
    Iby_FILL :	BYTE;
    Iby_ATTR :	BYTE;
    Iin_BORDER :	INT;
  END_VAR

  VAR_IN_OUT
    Xus_TN_SCREEN :	us_TN_SCREEN;
  END_VAR

  IF TN_SC_XY2_ERROR(Iin_X1,Iin_Y1,Iin_X2,Iin_Y2) THEN RETURN; END_IF;

  CASE Iin_Border OF
  0:
    in_Border_Offset := 0;

  1:
    by_BorderCHAR_L_T := BYTE#218;
    by_BorderCHAR_T   := BYTE#196;
    by_BorderCHAR_R_T := BYTE#191;
    by_BorderCHAR_L   := BYTE#179;
    by_BorderCHAR_R   := BYTE#179;
    by_BorderCHAR_B   := BYTE#196;
    by_BorderCHAR_L_B := BYTE#217;
    by_BorderCHAR_R_B := BYTE#192;
    in_Border_Offset  := 1;

  2:
    by_BorderCHAR_L_T := BYTE#201;
    by_BorderCHAR_T   := BYTE#205;
    by_BorderCHAR_R_T := BYTE#187;
    by_BorderCHAR_L   := BYTE#186;
    by_BorderCHAR_R   := BYTE#186;
    by_BorderCHAR_B   := BYTE#205;
    by_BorderCHAR_L_B := BYTE#188;
    by_BorderCHAR_R_B := BYTE#200;
    in_Border_Offset  := 1;

  ELSE
    by_BorderCHAR_L_T := BYTE#32;
    by_BorderCHAR_T   := BYTE#32;
    by_BorderCHAR_R_T := BYTE#32;
    by_BorderCHAR_L   := BYTE#32;
    by_BorderCHAR_R   := BYTE#32;
    by_BorderCHAR_B   := BYTE#32;
    by_BorderCHAR_L_B := BYTE#32;
    by_BorderCHAR_R_B := BYTE#32;
    in_Border_Offset  := 1;

  END_CASE;

  IF Iby_FILL > BYTE#0 THEN

    FB_TN_SC_FILL.Iin_Y1			:= Iin_Y1 + in_Border_Offset;
    FB_TN_SC_FILL.Iin_X1			:= Iin_X1 + in_Border_Offset;
    FB_TN_SC_FILL.Iin_Y2			:= Iin_Y2 - in_Border_Offset;
    FB_TN_SC_FILL.Iin_X2			:= Iin_X2 - in_Border_Offset;
    FB_TN_SC_FILL.Iby_CHAR		:= Iby_FILL;
    FB_TN_SC_FILL.Iby_Attr		:= Iby_ATTR;
    FB_TN_SC_FILL.Xus_TN_SCREEN := Xus_TN_SCREEN;
    FB_TN_SC_FILL();
    Xus_TN_SCREEN := FB_TN_SC_FILL.Xus_TN_SCREEN;

  END_IF;

  IF Iin_BORDER = 0 THEN RETURN; END_IF;

  in_Offset_1 := (Iin_Y1 * 80) + Iin_X1;
  in_Offset_2 := (Iin_Y1 * 80) + Iin_X2;

  FOR in_Y := Iin_Y1 TO Iin_Y2 DO

    Xus_TN_SCREEN.bya_Line_Update[in_Y] := TRUE;

    Xus_TN_SCREEN.bya_CHAR[in_Offset_1]  := by_BorderCHAR_L;
    Xus_TN_SCREEN.bya_COLOR[in_Offset_1] := Iby_Attr;

    Xus_TN_SCREEN.bya_CHAR[in_Offset_2]  := by_BorderCHAR_R;
    Xus_TN_SCREEN.bya_COLOR[in_Offset_2] := Iby_Attr;

    in_Offset_1 := in_Offset_1 + 80;
    in_Offset_2 := in_Offset_2 + 80;

  END_FOR;

  in_Offset_1 := (Iin_Y1 * 80) + Iin_X1;
  in_Offset_2 := (Iin_Y2 * 80) + Iin_X1;

  FOR in_X := Iin_X1 TO Iin_X2 DO

    Xus_TN_SCREEN.bya_CHAR[in_Offset_1]  := by_BorderCHAR_T;
    Xus_TN_SCREEN.bya_COLOR[in_Offset_1] := Iby_Attr;

    Xus_TN_SCREEN.bya_CHAR[in_Offset_2]  := by_BorderCHAR_B;
    Xus_TN_SCREEN.bya_COLOR[in_Offset_2] := Iby_Attr;

    in_Offset_1 := in_Offset_1 + INT#1;
    in_Offset_2 := in_Offset_2 + INT#1;

  END_FOR;

  in_Offset_1 := (Iin_Y1 * 80) + Iin_X1;
  Xus_TN_SCREEN.bya_CHAR[in_Offset_1]  := by_BorderCHAR_L_T;
  Xus_TN_SCREEN.bya_COLOR[in_Offset_1] := Iby_Attr;

  in_Offset_1 := (Iin_Y1 * 80) + Iin_X2;
  Xus_TN_SCREEN.bya_CHAR[in_Offset_1]  := by_BorderCHAR_R_T;
  Xus_TN_SCREEN.bya_COLOR[in_Offset_1] := Iby_Attr;

  in_Offset_1 := (Iin_Y2 * 80) + Iin_X1;
  Xus_TN_SCREEN.bya_CHAR[in_Offset_1]  := by_BorderCHAR_R_B;
  Xus_TN_SCREEN.bya_COLOR[in_Offset_1] := Iby_Attr;

  in_Offset_1 := (Iin_Y2 * 80) + Iin_X2;
  Xus_TN_SCREEN.bya_CHAR[in_Offset_1]  := by_BorderCHAR_L_B;
  Xus_TN_SCREEN.bya_COLOR[in_Offset_1] := Iby_Attr;

END_FUNCTION_BLOCK

PROGRAM program0
	VAR
		Iin_Y1 :	INT;
    Iin_X1 :	INT;
    Iin_Y2 :	INT;
    Iin_X2 :	INT;
    Iby_FILL :	BYTE;
    Iby_ATTR :	BYTE;
    Iin_BORDER :	INT;
		Xus_TN_SCREEN :	us_TN_SCREEN;

		func_block : TN_SC_BOX_Block;
	END_VAR
  func_block.Iin_X1 := Iin_X1;
  func_block.Iin_Y1 := Iin_Y1;
  func_block.Iin_X2 := Iin_X2;
  func_block.Iin_Y2 := Iin_Y2;
  func_block.Iby_FILL := Iby_FILL;
  func_block.Iby_ATTR := Iby_ATTR;
  func_block.Iin_BORDER := Iin_BORDER;
  func_block.Xus_TN_SCREEN := Xus_TN_SCREEN;

	func_block();
	Xus_TN_SCREEN  := func_block.Xus_TN_SCREEN;
END_PROGRAM

CONFIGURATION Config0
	RESOURCE ReS0 ON PLC
		TASK task0(INTERVAL := T#20ms,PRIORITY := 0);
		PROGRAM instance0 WITH task0 : program0;
	END_RESOURCE
END_CONFIGURATION

(* ---- lb_claude_assisted_f2c634533beb_0043.st ---- *)
FUNCTION UDINT_TO_TIME2:TIME

	VAR_INPUT
		IN :	UDINT;
	END_VAR

	UDINT_TO_TIME2 := DINT_TO_TIME(UDINT_TO_DINT(IN));

END_FUNCTION

FUNCTION_BLOCK T_PLC_MS_block
	VAR_OUTPUT
		T_PLC_MS :	UDINT;
	END_VAR

	VAR_EXTERNAL
		PLC_TICKS_PER_SEC :	INT;
		PLC_SYS_TICK_CNT :	DINT;
	END_VAR

	VAR
		debug :	BOOL;
		N :	INT;
		Offset :	UDINT;
		temp :	DWORD := DWORD#1;
		mode :	BOOL;
		faktor :	UDINT;
		init :	BOOL;
		v_plc_ticks_per_sec :	UDINT;
		base :	UDINT := UDINT#1000;
	END_VAR

	IF init = FALSE THEN
		v_plc_ticks_per_sec := INT_TO_UDINT(PLC_TICKS_PER_SEC);
		IF v_plc_ticks_per_sec = UDINT#1024 THEN
			faktor := UDINT#1;
			mode := FALSE;
		ELSIF v_plc_ticks_per_sec > UDINT#0 THEN
			IF v_plc_ticks_per_sec <= base THEN
				faktor := base / v_plc_ticks_per_sec;
				mode := FALSE;
			ELSE
				faktor := v_plc_ticks_per_sec / base;
				mode := TRUE;
			END_IF;
		ELSE
			faktor := UDINT#1;
		END_IF;
		init := TRUE;
	END_IF;

	IF mode THEN
		T_PLC_MS := DINT_TO_UDINT(PLC_SYS_TICK_CNT) / faktor;
	ELSE
		T_PLC_MS := DINT_TO_UDINT(PLC_SYS_TICK_CNT) * faktor;
	END_IF;

	IF debug THEN
		T_PLC_MS := (DWORD_TO_UDINT(SHL(UDINT_TO_DWORD(T_PLC_MS),N) OR SHL(temp,N)) - UDINT#1) + Offset;
	END_IF;

END_FUNCTION_BLOCK

FUNCTION_BLOCK SEQUENCE_4_Block

	VAR_INPUT
		IN0 :	BOOL := TRUE;
		IN1 :	BOOL := TRUE;
		IN2 :	BOOL := TRUE;
		IN3 :	BOOL := TRUE;
		START :	BOOL;
		RST :	BOOL;
		WAIT0 :	TIME;
		DELAY0 :	TIME;
		WAIT1 :	TIME;
		DELAY1 :	TIME;
		WAIT2 :	TIME;
		DELAY2 :	TIME;
		WAIT3 :	TIME;
		DELAY3 :	TIME;
		STOP_ON_ERROR :	BOOL;
	END_VAR

	VAR_OUTPUT
		Q0 :	BOOL;
		Q1 :	BOOL;
		Q2 :	BOOL;
		Q3 :	BOOL;
		QX :	BOOL;
		RUN :	BOOL;
		_STEP :	INT := -1;
		STATUS :	BYTE;
	END_VAR

	VAR
		last :	TIME;
		edge :	BOOL;
		tx :	TIME;
		init :	BOOL;
		T_PLC_MS :	T_PLC_MS_Block;
	END_VAR

	T_PLC_MS();
	tx:= UDINT_TO_TIME(T_PLC_MS.T_PLC_MS);

	IF NOT init THEN
		last := tx;
		init := TRUE;
		status := BYTE#110;
	END_IF;

	IF rst THEN
		_step := -1;
		Q0 := FALSE;
		Q1 := FALSE;
		Q2 := FALSE;
		Q3 := FALSE;
		status := BYTE#110;
		run := FALSE;

	ELSIF start AND NOT edge THEN
		_step := 0;
		last := tx;
		status := BYTE#111;
		Q0 := FALSE;
		Q1 := FALSE;
		Q2 := FALSE;
		Q3 := FALSE;
		run := TRUE;
	END_IF;
	edge := start;

	IF status > BYTE#0 AND status < BYTE#100 AND stop_on_error THEN RETURN; END_IF;

	IF run AND _step = 0 THEN
		IF NOT q0 AND in0 AND tx - last <= wait0 THEN
			Q0 := TRUE;
			last := tx;
		ELSIF NOT q0 AND tx - last > wait0 THEN
			status := BYTE#1;
			run := FALSE;
		ELSIF q0 AND tx - last >= delay0 THEN
			_step := 1;
			last := tx;
		END_IF;
	END_IF;
	IF run AND _step = 1 THEN
		IF NOT q1 AND in1 AND tx - last <= wait1 THEN
			Q0 := FALSE;
			Q1 := TRUE;
			last := tx;
		ELSIF NOT q1 AND Tx - last > wait1 THEN
			status := BYTE#2;
			q0 := FALSE;
			run := FALSE;
		ELSIF q1 AND tx - last >= delay1 THEN
			_step := 2;
			last := tx;
		END_IF;
	END_IF;
	IF run AND _step = 2 THEN
		IF NOT q2 AND in2 AND tx - last <= wait2 THEN
			Q1 := FALSE;
			Q2 := TRUE;
			last := tx;
		ELSIF NOT q2 AND Tx - last > wait2 THEN
			status := BYTE#3;
			q1 := FALSE;
			run := FALSE;
		ELSIF q2 AND tx - last >= delay2 THEN
			_step := 3;
			last := tx;
		END_IF;
	END_IF;
	IF run AND _step = 3 THEN
		IF NOT q3 AND in3 AND tx - last <= wait3 THEN
			Q2 := FALSE;
			Q3 := TRUE;
			last := tx;
		ELSIF NOT q3 AND Tx - last > wait3 THEN
			status := BYTE#4;
			q2 := FALSE;
			run := FALSE;
		ELSIF q3 AND tx - last >= delay3 THEN
			_step := -1;
			q3 := FALSE;
			run := FALSE;
			status := BYTE#110;
		END_IF;
	END_IF;
	QX := q0 OR q1 OR q2 OR q3;

END_FUNCTION_BLOCK

PROGRAM program0

	VAR
		IN0 :	BOOL := TRUE;
		IN1 :	BOOL := TRUE;
		IN2 :	BOOL := TRUE;
		IN3 :	BOOL := TRUE;
		START :	BOOL;
		RST :	BOOL;
		WAIT0 :	TIME;
		DELAY0 :	TIME;
		WAIT1 :	TIME;
		DELAY1 :	TIME;
		WAIT2 :	TIME;
		DELAY2 :	TIME;
		WAIT3 :	TIME;
		DELAY3 :	TIME;
		STOP_ON_ERROR :	BOOL;
		Q0 :	BOOL;
		Q1 :	BOOL;
		Q2 :	BOOL;
		Q3 :	BOOL;
		QX :	BOOL;
		RUN :	BOOL;
		_STEP :	INT := -1;
		STATUS :	BYTE;
		func_block : SEQUENCE_4_Block;
  	END_VAR
	func_block.IN0  :=IN0;
	func_block.IN1  :=IN1;
	func_block.IN2  :=IN2;
	func_block.IN3  :=IN3;
	func_block.START  :=START;
	func_block.RST  :=RST;
	func_block.WAIT0  :=WAIT0;
	func_block.DELAY0  :=DELAY0;
	func_block.WAIT1:=WAIT1;
	func_block.DELAY1:=DELAY1;
	func_block.WAIT2  :=WAIT2;
	func_block.DELAY2  :=DELAY2;
	func_block.WAIT3  :=WAIT3;
	func_block.DELAY3  :=DELAY3;
	func_block.DELAY1:=DELAY1;
	func_block.WAIT2  :=WAIT2;
	func_block.DELAY2  :=DELAY2;
	func_block.WAIT3  :=WAIT3;
	func_block.DELAY3  :=DELAY3;
	func_block.STOP_ON_ERROR  :=STOP_ON_ERROR;
	func_block();
	Q0 := func_block.Q0;
	Q1 := func_block.Q1;
	Q2 := func_block.Q2;
	Q3 := func_block.Q3;
	QX := func_block.QX;
	RUN := func_block.RUN;
	_STEP := func_block._STEP;
	STATUS := func_block.STATUS;

END_PROGRAM

CONFIGURATION Config0

	VAR_GLOBAL
		PLC_TICKS_PER_SEC :	INT;
		PLC_SYS_TICK_CNT :	DINT;
	END_VAR

	RESOURCE Res0 ON PLC
		TASK task0(INTERVAL := T#20ms,PRIORITY := 0);
		PROGRAM instance0 WITH task0 : program0;
	END_RESOURCE

END_CONFIGURATION

(* ---- lb_claude_assisted_f3d1706a4ce0_0007.st ---- *)
FUNCTION_BLOCK T_PLC_MS_block
	VAR_OUTPUT
		T_PLC_MS :	UDINT;
	END_VAR

	VAR_EXTERNAL
		PLC_TICKS_PER_SEC :	INT;
		PLC_SYS_TICK_CNT :	DINT;
	END_VAR

	VAR
		debug :	BOOL;(*Debug-Mode ON / OFF*)
		N :	INT;(*Debug-Faktor*)
		Offset :	UDINT;(*Debug-Offset*)
		temp :	DWORD := DWORD#1;(*Debug-Offset*)
		mode :	BOOL;(*modus*)
		faktor :	UDINT;(*Systemtakt-Faktor*)
		init :	BOOL;
		v_plc_ticks_per_sec :	UDINT;
		base :	UDINT := UDINT#1000;
	END_VAR

	IF init = FALSE THEN
		v_plc_ticks_per_sec := INT_TO_UDINT(PLC_TICKS_PER_SEC);
		IF v_plc_ticks_per_sec = UDINT#1024 THEN
			faktor := UDINT#1;
			mode := FALSE;
		ELSIF v_plc_ticks_per_sec > UDINT#0 THEN
			IF v_plc_ticks_per_sec <= base THEN
				faktor := base / v_plc_ticks_per_sec;
				mode := FALSE;
			ELSE
				faktor := v_plc_ticks_per_sec / base;
				mode := TRUE;
			END_IF;
		ELSE
			faktor := UDINT#1;
		END_IF;
		init := TRUE;
	END_IF;

	IF mode THEN
		T_PLC_MS := DINT_TO_UDINT(PLC_SYS_TICK_CNT) / faktor;
	ELSE
		T_PLC_MS := DINT_TO_UDINT(PLC_SYS_TICK_CNT) * faktor;
	END_IF;

	IF debug THEN
		T_PLC_MS := (DWORD_TO_UDINT(SHL(UDINT_TO_DWORD(T_PLC_MS),N) OR SHL(temp,N)) - UDINT#1) + Offset;
	END_IF;

END_FUNCTION_BLOCK

FUNCTION_BLOCK ONTIME_Block

	VAR_INPUT
		IN :	BOOL;
		RST :	BOOL;
	END_VAR

	VAR_IN_OUT
		SECONDS :	UDINT;
		CYCLES :	UDINT;
	END_VAR

	VAR
		tx :	UDINT;
		last :	UDINT;
		edge :	BOOL;
		init :	BOOL;
		ms :	UDINT;
		T_PLC_MS :	T_PLC_MS_Block;
	END_VAR

	T_PLC_MS();
	tx:= T_PLC_MS.T_PLC_MS;

	IF NOT init THEN
		init := TRUE;
		last := tx;
		ms := UDINT#0;
	END_IF;
	IF RST THEN
		SECONDS := UDINT#0;
		CYCLES := UDINT#0;
		last := tx;
		ms := UDINT#0;
	ELSIF IN THEN
		(* add the current milliseconds *)
		ms := (tx - last) + ms;
		IF ms >= UDINT#1000 THEN
			seconds := seconds + UDINT#1;
			ms := ms - UDINT#1000;
		END_IF;
		cycles := cycles + BOOL_TO_UDINT(NOT edge);
	END_IF;
	last := tx;
	edge := in;

END_FUNCTION_BLOCK

FUNCTION_BLOCK ACTUATOR_PUMP_Block

	VAR_INPUT
		IN :	BOOL;
		MANUAL :	BOOL;
		RST :	BOOL := FALSE;
		MIN_ONTIME :	TIME := T#10s;
		MIN_OFFTIME :	TIME := T#10s;
		RUN_EVERY :	TIME := T#10000m;
	END_VAR

	VAR_OUTPUT
		PUMP :	BOOL;
		RUNTIME :	UDINT;
		CYCLES :	UDINT;
	END_VAR

	VAR
		tx :	TIME;
		last_change :	TIME;
		meter :	ONTIME_Block;
		old_man :	BOOL;
		init :	BOOL;
		T_PLC_MS :	T_PLC_MS_Block;
	END_VAR

	T_PLC_MS();
	tx:= UDINT_TO_TIME(T_PLC_MS.T_PLC_MS);

	IF NOT init THEN
		init := TRUE;
		last_change := tx;
	ELSIF rst THEN
		rst := FALSE;
		runtime := UDINT#0;
		cycles := UDINT#0;
	ELSIF manual AND NOT pump AND NOT old_man THEN
		last_change := tx;
		pump := TRUE;
	ELSIF NOT manual AND old_man AND pump AND NOT in THEN
		last_change := tx;
		pump := FALSE;
	ELSIF in AND NOT pump AND tx - last_change >= min_offtime THEN
		last_change := tx;
		pump := TRUE;
	ELSIF pump AND NOT in AND NOT manual AND tx - last_change >= min_ontime THEN
		last_change := tx;
		pump := FALSE;
	ELSIF NOT pump AND (tx - last_change >= run_every) AND (run_every > T#0s) THEN
		last_change := tx;
		pump := TRUE;
	END_IF;

	meter(in := pump, SECONDS := runtime, CYCLES := cycles);
	cycles := meter.CYCLES;
	runtime := meter.SECONDS;

	old_man := manual;

END_FUNCTION_BLOCK

PROGRAM program0
	VAR
		IN :	BOOL;
		MANUAL :	BOOL;
		RST :	BOOL := FALSE;
		MIN_ONTIME :	TIME := T#10s;
		MIN_OFFTIME :	TIME := T#10s;
		RUN_EVERY :	TIME := T#10000m;
		PUMP :	BOOL;
		RUNTIME :	UDINT;
		CYCLES :	UDINT;
		func_block : ACTUATOR_PUMP_Block;
	END_VAR
	func_block.IN := IN;
	func_block.MANUAL := MANUAL;
	func_block.RST := RST ;
	func_block.MIN_ONTIME := MIN_ONTIME;
	func_block.MIN_OFFTIME := MIN_OFFTIME;
	func_block.RUN_EVERY := RUN_EVERY ;
	func_block();
	PUMP  := func_block.PUMP;
	RUNTIME  := func_block.RUNTIME;
	CYCLES  := func_block.CYCLES;
END_PROGRAM

CONFIGURATION Config0
	VAR_GLOBAL
		PLC_TICKS_PER_SEC :	INT;
		PLC_SYS_TICK_CNT :	DINT;
	END_VAR
  	RESOURCE Res0 ON PLC
    	TASK task0(INTERVAL := T#20ms,PRIORITY := 0);
    	PROGRAM instance0 WITH task0 : program0;
  	END_RESOURCE
END_CONFIGURATION

(* ---- lb_claude_assisted_f6580cc4f869_0034.st ---- *)
FUNCTION_BLOCK T_PLC_MS_block
	VAR_OUTPUT
		T_PLC_MS :	UDINT;
	END_VAR

	VAR
		PLC_TICKS_PER_SEC :	INT;
		PLC_SYS_TICK_CNT :	DINT;
	END_VAR

	VAR
		debug :	BOOL;(*Debug-Mode ON / OFF*)
		N :	INT;(*Debug-Faktor*)
		Offset :	UDINT;(*Debug-Offset*)
		temp :	DWORD := DWORD#1;(*Debug-Offset*)
		MODE :	BOOL;(*modus*)
		faktor :	UDINT;(*Systemtakt-Faktor*)
		init :	BOOL;
		v_plc_ticks_per_sec :	UDINT;
		base :	UDINT := UDINT#1000;
	END_VAR

	IF init = FALSE THEN
		v_plc_ticks_per_sec := INT_TO_UDINT(PLC_TICKS_PER_SEC);
		IF v_plc_ticks_per_sec = UDINT#1024 THEN
			faktor := UDINT#1;
			MODE := FALSE;
		ELSIF v_plc_ticks_per_sec > UDINT#0 THEN
			IF v_plc_ticks_per_sec <= base THEN
				faktor := base / v_plc_ticks_per_sec;
				MODE := FALSE;
			ELSE
				faktor := v_plc_ticks_per_sec / base;
				MODE := TRUE;
			END_IF;
		ELSE
			faktor := UDINT#1;
		END_IF;
		init := TRUE;
	END_IF;

	IF MODE THEN
		T_PLC_MS := DINT_TO_UDINT(PLC_SYS_TICK_CNT) / faktor;
	ELSE
		T_PLC_MS := DINT_TO_UDINT(PLC_SYS_TICK_CNT) * faktor;
	END_IF;

	IF debug THEN
		T_PLC_MS := (DWORD_TO_UDINT(SHL(UDINT_TO_DWORD(T_PLC_MS),N) OR SHL(temp,N)) - UDINT#1) + Offset;
	END_IF;
END_FUNCTION_BLOCK

FUNCTION_BLOCK FT_RMP

	VAR_INPUT
		RMP :	BOOL := TRUE;
		IN :	REAL;
		KR :	REAL;
		KF :	REAL;
	END_VAR

	VAR_OUTPUT
		OUT :	REAL;
		BUSY :	BOOL;
		UD :	BOOL;
	END_VAR

	VAR
		TX :	TIME;
		last :	TIME;
		init :	BOOL;
		T_PLC_MS :	T_PLC_MS_block;
	END_VAR

	T_PLC_MS();
	TX:= SUB_TIME(UDINT_TO_TIME(T_PLC_MS.T_PLC_MS), last);

	IF NOT init THEN
		init := TRUE;
		last := TX;
		TX := t#0s;
		OUT := IN;
	END_IF;
	IF NOT RMP THEN
		OUT := IN;
		BUSY := FALSE;
	ELSIF OUT > IN THEN
		(* ramp down *)
		OUT := OUT - TIME_TO_REAL(TX) * 0.001 * KF;
		OUT := MAX(IN, OUT);
	ELSIF OUT < IN THEN
		(* ramp up *)
		OUT := OUT + TIME_TO_REAL(TX) * 0.001 * KR;
		OUT := MIN(IN, OUT);
	END_IF;

	(* set BUSY and DIR flags *)
	IF OUT < IN THEN
		BUSY := TRUE;
		UD := TRUE;
	ELSIF OUT > IN THEN
		BUSY := TRUE;
		UD := FALSE;
	ELSE
		BUSY := FALSE;
	END_IF;
	last := ADD_TIME(last, TX);

END_FUNCTION_BLOCK

PROGRAM program0
	VAR
		RMP :	BOOL := TRUE;
		IN :	REAL;
		KR :	REAL;
		KF :	REAL;

		OUT :	REAL;
		BUSY :	BOOL;
		UD :	BOOL;

		func_block : FT_RMP;
	END_VAR
	func_block.RMP := RMP;
	func_block.IN := IN;
	func_block.KR := KR;
	func_block.KF := KF;
	func_block();
	OUT := func_block.OUT;
	BUSY := func_block.BUSY;
	UD := func_block.UD;

END_PROGRAM

(* ---- lb_claude_assisted_f98caebf3a59_0014.st ---- *)
TYPE
  LOGLEVEL : (CRITICAL, WARNING, INFO, DEBUG) := INFO;
END_TYPE

FUNCTION_BLOCK LOGGER
  VAR_INPUT
    TRIG : BOOL;
    MSG : STRING;
    LEVEL : LOGLEVEL := INFO;
  END_VAR
  VAR
    TRIG0 : BOOL;
  END_VAR

  IF TRIG AND NOT TRIG0 THEN
  {{
   LogMessage(GetFbVar(LEVEL),(char*)GetFbVar(MSG, .body),GetFbVar(MSG, .len));
  }}
  END_IF;
  TRIG0:=TRIG;
END_FUNCTION_BLOCK

PROGRAM Paletizador
  VAR
    Inicio : BOOL;
    Paro : BOOL;
    Motor_cinta_Horizontal : BOOL;
    Motor_cinta_Inclinado : BOOL;
    Motor_cinta_Paletizador : BOOL;
    Contador_Cajas : BOOL;
    Piston_1 : BOOL;
    Sensor_Piston_1 : BOOL;
  END_VAR
  VAR
    CTU0 : CTU;
  END_VAR
  VAR
    Piston_Compuerta : BOOL;
    Sensor_Piston_Compuerta : BOOL;
    Compuerta : BOOL;
    Sensor_Compuerta : BOOL;
  END_VAR
  VAR
    CTU1 : CTU;
  END_VAR
  VAR
    Generador_Cajas : BOOL;
  END_VAR
  VAR
    TON0 : TON;
    Retardo : TIME := T#1000ms;
  END_VAR
  VAR
    Cinta_Pale0 : BOOL;
    Cinta_Pale1 : BOOL;
    Generador_pales : BOOL;
    Cinta_Paletizador : BOOL;
    Sensor_Pale_0 : BOOL;
    Sensor_Pale_1 : BOOL;
    limite_altura : BOOL;
    subir_pale : BOOL;
    bajar_pale : BOOL;
  END_VAR
  VAR
    TOF0 : TOF;
    TOF1 : TOF;
    TON1 : TON;
  END_VAR
  VAR
    Sensor_Pales : BOOL;
    sensor_ascensor : BOOL;
  END_VAR
  VAR
    CTU2 : CTU;
    TON2 : TON;
  END_VAR
  VAR
    sensor_bajada : BOOL;
  END_VAR
  VAR
    TON3 : TON;
    TOF2 : TOF;
    TON4 : TON;
    R_TRIG1 : R_TRIG;
    R_TRIG2 : R_TRIG;
    R_TRIG3 : R_TRIG;
    R_TRIG4 : R_TRIG;
    R_TRIG5 : R_TRIG;
    R_TRIG6 : R_TRIG;
    R_TRIG7 : R_TRIG;
    R_TRIG8 : R_TRIG;
    R_TRIG9 : R_TRIG;
    R_TRIG10 : R_TRIG;
  END_VAR

  Motor_cinta_Horizontal := NOT(Paro) AND (Generador_Cajas OR Inicio OR Motor_cinta_Horizontal OR Motor_cinta_Inclinado OR Motor_cinta_Paletizador);
  Motor_cinta_Inclinado := NOT(Paro) AND (Generador_Cajas OR Inicio OR Motor_cinta_Horizontal OR Motor_cinta_Inclinado OR Motor_cinta_Paletizador);
  Motor_cinta_Paletizador := NOT(Paro) AND (Generador_Cajas OR Inicio OR Motor_cinta_Horizontal OR Motor_cinta_Inclinado OR Motor_cinta_Paletizador);
  R_TRIG1(CLK := Contador_Cajas);
  R_TRIG2(CLK := Sensor_Piston_1);
  CTU0(CU := R_TRIG1.Q, R := R_TRIG2.Q, PV := 2);
  Piston_1 := CTU0.Q;
  R_TRIG3(CLK := Contador_Cajas);
  CTU1(CU := R_TRIG3.Q, R := Sensor_Piston_Compuerta, PV := 6);
  TON0(IN := CTU1.Q, PT := Retardo);
  Piston_Compuerta := TON0.Q;
  Sensor_Piston_Compuerta := Sensor_Piston_Compuerta;
  Generador_Cajas := NOT(Paro) AND (Generador_Cajas OR Inicio OR Motor_cinta_Horizontal OR Motor_cinta_Inclinado OR Motor_cinta_Paletizador);
  Sensor_Piston_1 := NOT(NOT(Sensor_Piston_1));
  TOF1(IN := Sensor_Piston_Compuerta, PT := T#3500ms);
  Compuerta := TOF1.Q;
  TON1(IN := Sensor_Pales, PT := T#2000ms);
  TOF0(IN := TON1.Q, PT := T#3500ms);
  subir_pale := TOF0.Q;
  limite_altura := TOF0.Q;
  bajar_pale := Compuerta;
  R_TRIG4(CLK := sensor_ascensor);
  TON3(IN := sensor_bajada, PT := T#2000ms);
  CTU2(CU := R_TRIG4.Q, R := TON3.Q, PV := 3);
  TON2(IN := CTU2.Q, PT := T#2000ms);
  IF TON2.Q THEN
    limite_altura := TRUE; (*set*)
  END_IF;
  IF TON2.Q THEN
    bajar_pale := TRUE; (*set*)
  END_IF;
  R_TRIG5(CLK := sensor_bajada);
  Cinta_Pale0 := NOT(Paro) AND (Cinta_Pale0 OR Cinta_Pale1 OR Cinta_Paletizador OR Generador_pales OR Inicio OR sensor_ascensor AND R_TRIG5.Q);
  R_TRIG6(CLK := sensor_bajada);
  Cinta_Pale1 := NOT(Paro) AND (Cinta_Pale0 OR Cinta_Pale1 OR Cinta_Paletizador OR Generador_pales OR Inicio OR sensor_ascensor AND R_TRIG6.Q);
  R_TRIG7(CLK := sensor_bajada);
  Cinta_Paletizador := NOT(Paro) AND (Cinta_Pale0 OR Cinta_Pale1 OR Cinta_Paletizador OR Generador_pales OR Inicio OR sensor_ascensor AND R_TRIG7.Q);
  R_TRIG8(CLK := sensor_bajada);
  Generador_pales := NOT(Paro) AND (Cinta_Pale0 OR Cinta_Pale1 OR Cinta_Paletizador OR Generador_pales OR Inicio OR sensor_ascensor AND R_TRIG8.Q);
  TOF2(IN := Sensor_Pales, PT := T#3700ms);
  TON4(IN := TOF2.Q, PT := T#3700ms);
  IF TON4.Q THEN
    Cinta_Pale0 := FALSE; (*reset*)
  END_IF;
  IF TON4.Q THEN
    Cinta_Pale1 := FALSE; (*reset*)
  END_IF;
  IF TON4.Q THEN
    Cinta_Paletizador := FALSE; (*reset*)
  END_IF;
  IF TON4.Q THEN
    Generador_pales := FALSE; (*reset*)
  END_IF;
  R_TRIG9(CLK := sensor_bajada);
  IF NOT(Paro) AND (Cinta_Pale0 OR Cinta_Pale1 OR Cinta_Paletizador OR Generador_pales OR Inicio OR sensor_ascensor AND R_TRIG9.Q) THEN
    limite_altura := FALSE; (*reset*)
  END_IF;
  R_TRIG10(CLK := sensor_bajada);
  IF NOT(Paro) AND (Cinta_Pale0 OR Cinta_Pale1 OR Cinta_Paletizador OR Generador_pales OR Inicio OR sensor_ascensor AND R_TRIG10.Q) THEN
    bajar_pale := FALSE; (*reset*)
  END_IF;
END_PROGRAM

CONFIGURATION Config0

  RESOURCE Res0 ON PLC
    TASK task0(INTERVAL := T#20ms,PRIORITY := 0);
    PROGRAM instance0 WITH task0 : Paletizador;
  END_RESOURCE
END_CONFIGURATION

(* ---- lb_claude_assisted_fa801b45c55f_0059.st ---- *)
(*
This code implements a randomly grown symbolic expression:

!(((xor(xor(((!((xor(xor(IN5 & IN31, IN14), xor(xor(IN41, IN34), IN36))) | (xor(xor(IN5 & true, xor(xor(IN20, IN11), IN46)), xor(xor(IN9, IN25), IN28))))) | ((!((IN16 | IN46) | (IN34 | IN14))) & (((!(IN2)) & (IN5 | IN10)) | (xor(xor(xor(xor(IN46, IN24), IN5), IN28), xor(xor(IN22, IN7), IN13)))))) | (!(IN19 | (xor(xor((!(IN12)) | (IN2 & IN50), IN16), (IN45 & IN28) & IN21)))), xor(xor((xor(xor((xor(xor(IN6 & IN27, IN43 | IN5), IN28)) | (!(IN20 | IN22)), (IN35 & (IN50 | IN10)) | (!(IN19 & IN2))), IN7)) & (!(xor(xor((IN40 | IN16) & (xor(xor(IN27, IN8), IN19)), (xor(xor(IN45, IN13), IN13)) | (IN25 | IN3)), xor(xor(!(IN49), IN29 & IN12), IN16)))), ((!(xor(xor(xor(xor(IN33, IN26), IN50), !(IN42)), !(IN30)))) & IN3) & (xor(xor(!(xor(xor(IN2, xor(xor(false, IN16), true)), xor(xor(IN17, IN11), IN10))), IN24), ((IN41 | IN26) & (!(IN44))) & (!(!(IN6)))))), IN30 & IN4)), xor(xor(xor(xor(!((xor(xor(xor(xor(IN31, IN12), IN9), IN26 | IN38), xor(xor(IN20, IN24), IN46))) | ((IN20 & true) & IN13)), (!(IN36)) | (xor(xor(xor(xor(xor(xor(IN2, IN48), IN8), xor(xor(IN24, IN16), IN9)), IN50 & IN17), IN49), (xor(xor(IN31, true), IN31)) | (xor(xor(IN16, IN38), IN3))))), IN32), IN39), xor(xor((IN17 & (xor(xor(IN35, IN17), !(IN22)))) & (!((!(IN41)) | (IN28 | true))), xor(xor(((!(IN13)) & (xor(xor(IN29, IN36), IN8))) | (xor(xor(IN23 | IN37, IN18 | IN30), IN14 & IN24)), IN39), IN35)), (((IN5 | IN5) & (xor(xor(IN38, IN9), IN45))) & (xor(xor(xor(xor(IN14, IN9), IN1), xor(xor(IN3, IN7), IN34)), !(IN5)))) & ((xor(xor(true | IN3, IN49), IN17 | IN7)) | (!(xor(xor(IN29, IN5), IN48)))))))) | ((xor(xor(xor(xor(xor(xor(!((xor(xor(IN22, IN48), IN22)) | (xor(xor(IN2, true), IN15))), !(IN23)), false), !(((!(IN29)) | (IN46 & IN10)) & ((IN43 | IN35) & IN45))), IN5), (((!(IN35 & true)) | IN22) | (IN39 & (xor(xor(!(IN23), !(IN14)), IN5)))) | (false & (((true & IN42) | (xor(xor(IN16, IN12), IN19))) & (xor(xor(IN5 | IN16, !(IN31)), IN13 & IN46))))), xor(xor(((xor(xor(false & IN31, !(IN12)), IN38)) | ((IN12 & IN14) & IN26)) | (IN14 & (xor(xor(IN42 | IN16, IN50 | IN20), IN1 | IN31))), ((xor(xor(IN44 & IN16, IN29 & IN26), IN19)) & (xor(xor(IN17 & IN46, !(IN42)), xor(xor(IN40, IN42), IN9)))) & ((xor(xor(IN16, !(IN41)), IN2 & IN40)) | ((IN36 | IN3) | IN49))), ((xor(xor(IN35 & IN9, IN19 & IN34), IN12 | IN47)) & ((IN45 & IN19) & (!(IN33)))) | (((IN40 | IN32) | (IN2 | true)) & (xor(xor(IN40 & IN15, xor(xor(IN30, IN5), IN35)), IN48 & IN16)))))) & (!((xor(xor(IN16, IN15), !(!(true & IN45)))) & ((((!(IN44)) | (IN16 & IN26)) | IN43) | (((xor(xor(IN42, IN39), IN40)) | (IN42 & IN8)) & (xor(xor(IN37 & IN7, !(IN1)), IN30 | IN24)))))))) | (!(IN24)))

*)

FUNCTION_BLOCK F_CollectInput
  VAR_IN_OUT
      Data : ARRAY[1..50] OF BOOL;
  END_VAR
  VAR_INPUT
      TICK  : BOOL := 0;
      IN1   : BOOL := 0;
      IN2   : BOOL := 0;
      IN3   : BOOL := 0;
      IN4   : BOOL := 0;
      IN5   : BOOL := 0;
      RESET : BOOL := FALSE;
  END_VAR
  VAR_OUTPUT
      Finished : BOOL;
  END_VAR
  VAR
      j    : USINT := 1;
      tock : BOOL  := 0;
  END_VAR
  IF NOT RESET AND tock = NOT TICK THEN
      Data[j]   := IN1;
      Data[j+1] := IN2;
      Data[j+2] := IN3;
      Data[j+3] := IN4;
      Data[j+4] := IN5;
      j := j + 5;
      tock := TICK;
  ELSE
      j := 1;
      tock := 0;
  END_IF;
  Finished := (j > 50);
END_FUNCTION_BLOCK

PROGRAM Boiler
  VAR
    Data  : ARRAY[1..50] OF BOOL;
    Ready : BOOL;
    CollectInput : F_CollectInput;
  END_VAR
  VAR
    TICK     AT %IX1.0 : BOOL;
    IN1      AT %IX0.3 : BOOL;
    IN2      AT %IX0.4 : BOOL;
    IN3      AT %IX0.5 : BOOL;
    IN4      AT %IX0.6 : BOOL;
    IN5      AT %IX0.7 : BOOL;
    OutReady AT %QX0.0 : BOOL := FALSE;
    FeedNext AT %QX0.1 : BOOL := FALSE;
    Out      AT %QX0.2 : BOOL;
  END_VAR
  CollectInput(TICK:=TICK, IN1:=IN1, IN2:=IN2, IN3:=IN3, IN4:=IN4, IN5:=IN5);
  Ready := CollectInput.Finished;
  FeedNext := 1;
  IF Ready THEN
    Out := (NOT (((((((NOT ((((Data[5] AND Data[31]) XOR Data[14]) XOR ((Data[41] XOR Data[34]) XOR Data[36])) OR (((Data[5] AND TRUE) XOR ((Data[20] XOR Data[11]) XOR Data[46])) XOR ((Data[9] XOR Data[25]) XOR Data[28])))) OR ((NOT ((Data[16] OR Data[46]) OR (Data[34] OR Data[14]))) AND (((NOT Data[2]) AND (Data[5] OR Data[10])) OR ((((Data[46] XOR Data[24]) XOR Data[5]) XOR Data[28]) XOR ((Data[22] XOR Data[7]) XOR Data[13]))))) OR (NOT (Data[19] OR ((((NOT Data[12]) OR (Data[2] AND Data[50])) XOR Data[16]) XOR ((Data[45] AND Data[28]) AND Data[21]))))) XOR (((((((((Data[6] AND Data[27]) XOR (Data[43] OR Data[5])) XOR Data[28]) OR (NOT (Data[20] OR Data[22]))) XOR ((Data[35] AND (Data[50] OR Data[10])) OR (NOT (Data[19] AND Data[2])))) XOR Data[7]) AND (NOT ((((Data[40] OR Data[16]) AND ((Data[27] XOR Data[8]) XOR Data[19])) XOR (((Data[45] XOR Data[13]) XOR Data[13]) OR (Data[25] OR Data[3]))) XOR (((NOT Data[49]) XOR (Data[29] AND Data[12])) XOR Data[16])))) XOR (((NOT ((((Data[33] XOR Data[26]) XOR Data[50]) XOR (NOT Data[42])) XOR (NOT Data[30]))) AND Data[3]) AND (((NOT ((Data[2] XOR ((FALSE XOR Data[16]) XOR TRUE)) XOR ((Data[17] XOR Data[11]) XOR Data[10]))) XOR Data[24]) XOR (((Data[41] OR Data[26]) AND (NOT Data[44])) AND (NOT (NOT Data[6])))))) XOR (Data[30] AND Data[4]))) XOR (((((NOT (((((Data[31] XOR Data[12]) XOR Data[9]) XOR (Data[26] OR Data[38])) XOR ((Data[20] XOR Data[24]) XOR Data[46])) OR ((Data[20] AND TRUE) AND Data[13]))) XOR ((NOT Data[36]) OR ((((((Data[2] XOR Data[48]) XOR Data[8]) XOR ((Data[24] XOR Data[16]) XOR Data[9])) XOR (Data[50] AND Data[17])) XOR Data[49]) XOR (((Data[31] XOR TRUE) XOR Data[31]) OR ((Data[16] XOR Data[38]) XOR Data[3]))))) XOR Data[32]) XOR Data[39]) XOR ((((Data[17] AND ((Data[35] XOR Data[17]) XOR (NOT Data[22]))) AND (NOT ((NOT Data[41]) OR (Data[28] OR TRUE)))) XOR (((((NOT Data[13]) AND ((Data[29] XOR Data[36]) XOR Data[8])) OR (((Data[23] OR Data[37]) XOR (Data[18] OR Data[30])) XOR (Data[14] AND Data[24]))) XOR Data[39]) XOR Data[35])) XOR ((((Data[5] OR Data[5]) AND ((Data[38] XOR Data[9]) XOR Data[45])) AND ((((Data[14] XOR Data[9]) XOR Data[1]) XOR ((Data[3] XOR Data[7]) XOR Data[34])) XOR (NOT Data[5]))) AND ((((TRUE OR Data[3]) XOR Data[49]) XOR (Data[17] OR Data[7])) OR (NOT ((Data[29] XOR Data[5]) XOR Data[48]))))))) OR ((((((((NOT (((Data[22] XOR Data[48]) XOR Data[22]) OR ((Data[2] XOR TRUE) XOR Data[15]))) XOR (NOT Data[23])) XOR FALSE) XOR (NOT (((NOT Data[29]) OR (Data[46] AND Data[10])) AND ((Data[43] OR Data[35]) AND Data[45])))) XOR Data[5]) XOR ((((NOT (Data[35] AND TRUE)) OR Data[22]) OR (Data[39] AND (((NOT Data[23]) XOR (NOT Data[14])) XOR Data[5]))) OR (FALSE AND (((TRUE AND Data[42]) OR ((Data[16] XOR Data[12]) XOR Data[19])) AND (((Data[5] OR Data[16]) XOR (NOT Data[31])) XOR (Data[13] AND Data[46])))))) XOR (((((((FALSE AND Data[31]) XOR (NOT Data[12])) XOR Data[38]) OR ((Data[12] AND Data[14]) AND Data[26])) OR (Data[14] AND (((Data[42] OR Data[16]) XOR (Data[50] OR Data[20])) XOR (Data[1] OR Data[31])))) XOR (((((Data[44] AND Data[16]) XOR (Data[29] AND Data[26])) XOR Data[19]) AND (((Data[17] AND Data[46]) XOR (NOT Data[42])) XOR ((Data[40] XOR Data[42]) XOR Data[9]))) AND (((Data[16] XOR (NOT Data[41])) XOR (Data[2] AND Data[40])) OR ((Data[36] OR Data[3]) OR Data[49])))) XOR (((((Data[35] AND Data[9]) XOR (Data[19] AND Data[34])) XOR (Data[12] OR Data[47])) AND ((Data[45] AND Data[19]) AND (NOT Data[33]))) OR (((Data[40] OR Data[32]) OR (Data[2] OR TRUE)) AND (((Data[40] AND Data[15]) XOR ((Data[30] XOR Data[5]) XOR Data[35])) XOR (Data[48] AND Data[16])))))) AND (NOT (((Data[16] XOR Data[15]) XOR (NOT (NOT (TRUE AND Data[45])))) AND ((((NOT Data[44]) OR (Data[16] AND Data[26])) OR Data[43]) OR ((((Data[42] XOR Data[39]) XOR Data[40]) OR (Data[42] AND Data[8])) AND (((Data[37] AND Data[7]) XOR (NOT Data[1])) XOR (Data[30] OR Data[24])))))))) OR (NOT Data[24])));
    OutReady := 1;
    CollectInput(RESET:=TRUE);
  END_IF;
END_PROGRAM

CONFIGURATION Config0
  RESOURCE Res0 ON PLC
    TASK task0(INTERVAL := T#20ms,PRIORITY := 0);
    PROGRAM instance0 WITH task0 : Boiler;
  END_RESOURCE
END_CONFIGURATION

(* ---- lb_claude_assisted_fcddad10f7fe_0048.st ---- *)
FUNCTION _REAL_TO_UDINT:UDINT
  VAR_INPUT
    X :	REAL;
  END_VAR

  IF REAL_TO_UDINT(0.5) = UDINT#1 THEN
    _REAL_TO_UDINT := REAL_TO_UDINT(x);
  ELSIF X > 0.0 THEN
    _REAL_TO_UDINT := REAL_TO_UDINT(x+0.5);
  ELSIF X < 0.0 THEN
    _REAL_TO_UDINT := REAL_TO_UDINT(x-0.5);
  ELSE
    _REAL_TO_UDINT := UDINT#0;
  END_IF;
END_FUNCTION

FUNCTION_BLOCK T_PLC_MS_block

	VAR_OUTPUT
		T_PLC_MS :	UDINT;
	END_VAR

	VAR_EXTERNAL
		PLC_TICKS_PER_SEC :	INT;
		PLC_SYS_TICK_CNT :	DINT;
	END_VAR

	VAR
		debug :	BOOL;(*Debug-Mode ON / OFF*)
		N :	INT;(*Debug-Faktor*)
		Offset :	UDINT;(*Debug-Offset*)
		temp :	DWORD := DWORD#1;(*Debug-Offset*)
		mode :	BOOL;(*modus*)
		faktor :	UDINT;(*Systemtakt-Faktor*)
		init :	BOOL;
		v_plc_ticks_per_sec :	UDINT;
		base :	UDINT := UDINT#1000;
	END_VAR

	IF init = FALSE THEN
		v_plc_ticks_per_sec := INT_TO_UDINT(PLC_TICKS_PER_SEC);
		IF v_plc_ticks_per_sec = UDINT#1024 THEN
			faktor := UDINT#1;
			mode := FALSE;
		ELSIF v_plc_ticks_per_sec > UDINT#0 THEN
			IF v_plc_ticks_per_sec <= base THEN
				faktor := base / v_plc_ticks_per_sec;
				mode := FALSE;
			ELSE
				faktor := v_plc_ticks_per_sec / base;
				mode := TRUE;
			END_IF;
		ELSE
			faktor := UDINT#1;
		END_IF;
		init := TRUE;
	END_IF;

	IF mode THEN
		T_PLC_MS := DINT_TO_UDINT(PLC_SYS_TICK_CNT) / faktor;
	ELSE
		T_PLC_MS := DINT_TO_UDINT(PLC_SYS_TICK_CNT) * faktor;
	END_IF;

	IF debug THEN
		T_PLC_MS := (DWORD_TO_UDINT(SHL(UDINT_TO_DWORD(T_PLC_MS),N) OR SHL(temp,N)) - UDINT#1) + Offset;
	END_IF;

END_FUNCTION_BLOCK

FUNCTION_BLOCK DT_SIMU
	VAR_INPUT
		START :	UDINT;
		SPEED :	REAL := 1.0;
	END_VAR

	VAR_OUTPUT
		DTS :	UDINT;
	END_VAR

	VAR
		tc :	UDINT;
		init :	BOOL;
		last :	UDINT;
		tx :	UDINT;
		td :	UDINT;
		T_PLC_MS :	T_PLC_MS_block;
	END_VAR

	T_PLC_MS();
	tx:= T_PLC_MS.T_PLC_MS;
	tc := _REAL_TO_UDINT(UDINT_TO_REAL(tx - last) * speed);

	IF NOT init THEN
		init := TRUE;
		DTS := Start;
		tc := UDINT#0;
		last := tx;
	ELSIF SPEED = 0.0 THEN
		DTS := DTS + UDINT#1;
	ELSIF tc >= UDINT#1000 THEN
		td := (tc / UDINT#1000) * UDINT#1000;
		DTS := DTS + td;
		last := last + _REAL_TO_UDINT(UDINT_TO_REAL(td) / speed);
	END_IF;
END_FUNCTION_BLOCK

PROGRAM program0
  VAR
    LocalVar0 : UDINT;
	LocalVar1 : REAL;
	LocalOUT  : UDINT;
	func_block : DT_SIMU;
  END_VAR
	func_block.START  := LocalVar0;
	func_block.SPEED  := LocalVar1;
	func_block();
	LocalOUT := func_block.DTS;
END_PROGRAM

CONFIGURATION Config0

	VAR_GLOBAL
		PLC_TICKS_PER_SEC :	INT;
		PLC_SYS_TICK_CNT :	DINT;
	END_VAR

  	RESOURCE Res0 ON PLC
    	TASK task0(INTERVAL := T#20ms,PRIORITY := 0);
    	PROGRAM instance0 WITH task0 : program0;
  	END_RESOURCE

END_CONFIGURATION
